EventTableEntry 8242: Group=, Trigger=conv1_buffer_upper_go_down 8243, Actions=[conv1_pallet_lifter_upper_up 8244], Comment=, ActivationMode=2, Cyclic=false
EventTableTriggerIO 8243: IOValue=[1], IRC5Controller=? -1, Operator=0, SignalSource=ALab_CellC_v1.0_4 5362
EventTableActionIO 8244: IOValue=[0], IRC5Controller=? -1, SignalTarget=ALab_CellC_v1.0_4 5362
EventTableEntry 8245: Group=, Trigger=conv1_buffer_upper_go_down 8246, Actions=[conv1_pallet_lifter_upper_up 8247], Comment=, ActivationMode=2, Cyclic=false
EventTableTriggerIO 8246: IOValue=[0], IRC5Controller=? -1, Operator=0, SignalSource=ALab_CellC_v1.0_4 5362
EventTableActionIO 8247: IOValue=[1], IRC5Controller=? -1, SignalTarget=ALab_CellC_v1.0_4 5362
EventTableEntry 8248: Group=, Trigger=conv1_buffer_upper_go_down 8249, Actions=[conv1_pallet_lifter_upper_down 8250], Comment=, ActivationMode=2, Cyclic=false
EventTableTriggerIO 8249: IOValue=[0], IRC5Controller=? -1, Operator=0, SignalSource=ALab_CellC_v1.0_4 5362
EventTableActionIO 8250: IOValue=[0], IRC5Controller=? -1, SignalTarget=ALab_CellC_v1.0_4 5362
EventTableEntry 8251: Group=, Trigger=conv1_buffer_upper_go_down 8252, Actions=[conv1_pallet_lifter_upper_down 8253], Comment=, ActivationMode=2, Cyclic=false
EventTableTriggerIO 8252: IOValue=[1], IRC5Controller=? -1, Operator=0, SignalSource=ALab_CellC_v1.0_4 5362
EventTableActionIO 8253: IOValue=[1], IRC5Controller=? -1, SignalTarget=ALab_CellC_v1.0_4 5362
EventTableEntry 8254: Group=, Trigger=conv1_buffer_lower_go_up 8255, Actions=[conv1_pallet_lifter_lower_down 8256], Comment=, ActivationMode=2, Cyclic=false
EventTableTriggerIO 8255: IOValue=[0], IRC5Controller=? -1, Operator=0, SignalSource=ALab_CellC_v1.0_4 5362
EventTableActionIO 8256: IOValue=[1], IRC5Controller=? -1, SignalTarget=ALab_CellC_v1.0_4 5362
EventTableEntry 8257: Group=, Trigger=conv1_buffer_lower_go_up 8258, Actions=[conv1_pallet_lifter_lower_down 8259], Comment=, ActivationMode=2, Cyclic=false
EventTableTriggerIO 8258: IOValue=[1], IRC5Controller=? -1, Operator=0, SignalSource=ALab_CellC_v1.0_4 5362
EventTableActionIO 8259: IOValue=[0], IRC5Controller=? -1, SignalTarget=ALab_CellC_v1.0_4 5362
EventTableEntry 8260: Group=, Trigger=conv2_buffer_horizontal_move 8261, Actions=[conv2_pallet_lifter_in 8262], Comment=, ActivationMode=2, Cyclic=false
EventTableTriggerIO 8261: IOValue=[1], IRC5Controller=? -1, Operator=0, SignalSource=ALab_CellC_v1.0_4 5362
EventTableActionIO 8262: IOValue=[1], IRC5Controller=? -1, SignalTarget=ALab_CellC_v1.0_4 5362
EventTableEntry 8263: Group=, Trigger=conv2_buffer_horizontal_move 8264, Actions=[conv2_pallet_lifter_in 8265], Comment=, ActivationMode=2, Cyclic=false
EventTableTriggerIO 8264: IOValue=[0], IRC5Controller=? -1, Operator=0, SignalSource=ALab_CellC_v1.0_4 5362
EventTableActionIO 8265: IOValue=[0], IRC5Controller=? -1, SignalTarget=ALab_CellC_v1.0_4 5362
EventTableEntry 8266: Group=, Trigger=conv2_buffer_horizontal_move 8267, Actions=[conv2_pallet_lifter_out 8268], Comment=, ActivationMode=2, Cyclic=false
EventTableTriggerIO 8267: IOValue=[0], IRC5Controller=? -1, Operator=0, SignalSource=ALab_CellC_v1.0_4 5362
EventTableActionIO 8268: IOValue=[1], IRC5Controller=? -1, SignalTarget=ALab_CellC_v1.0_4 5362
EventTableEntry 8269: Group=, Trigger=conv2_buffer_horizontal_move 8270, Actions=[conv2_pallet_lifter_out 8271], Comment=, ActivationMode=2, Cyclic=false
EventTableTriggerIO 8270: IOValue=[1], IRC5Controller=? -1, Operator=0, SignalSource=ALab_CellC_v1.0_4 5362
EventTableActionIO 8271: IOValue=[0], IRC5Controller=? -1, SignalTarget=ALab_CellC_v1.0_4 5362
EventTableEntry 8272: Group=, Trigger=conv2_buffer_lower_vertical_move 8273, Actions=[conv2_pallet_lifter_lower_down 8274], Comment=, ActivationMode=2, Cyclic=false
EventTableTriggerIO 8273: IOValue=[1], IRC5Controller=? -1, Operator=0, SignalSource=ALab_CellC_v1.0_4 5362
EventTableActionIO 8274: IOValue=[0], IRC5Controller=? -1, SignalTarget=ALab_CellC_v1.0_4 5362
EventTableEntry 8275: Group=, Trigger=conv2_buffer_lower_vertical_move 8276, Actions=[conv2_pallet_lifter_lower_down 8277], Comment=, ActivationMode=2, Cyclic=false
EventTableTriggerIO 8276: IOValue=[0], IRC5Controller=? -1, Operator=0, SignalSource=ALab_CellC_v1.0_4 5362
EventTableActionIO 8277: IOValue=[1], IRC5Controller=? -1, SignalTarget=ALab_CellC_v1.0_4 5362
EventTableEntry 8278: Group=, Trigger=conv2_buffer_upper_vertical_move 8279, Actions=[conv2_pallet_lifter_upper_up 8280], Comment=, ActivationMode=2, Cyclic=false
EventTableTriggerIO 8279: IOValue=[0], IRC5Controller=? -1, Operator=0, SignalSource=ALab_CellC_v1.0_4 5362
EventTableActionIO 8280: IOValue=[1], IRC5Controller=? -1, SignalTarget=ALab_CellC_v1.0_4 5362
EventTableEntry 8281: Group=, Trigger=conv2_buffer_upper_vertical_move 8282, Actions=[conv2_pallet_lifter_upper_up 8283], Comment=, ActivationMode=2, Cyclic=false
EventTableTriggerIO 8282: IOValue=[1], IRC5Controller=? -1, Operator=0, SignalSource=ALab_CellC_v1.0_4 5362
EventTableActionIO 8283: IOValue=[0], IRC5Controller=? -1, SignalTarget=ALab_CellC_v1.0_4 5362
EventTableEntry 8284: Group=, Trigger=conv2_buffer_upper_vertical_move 8285, Actions=[conv2_pallet_lifter_upper_down 8286], Comment=, ActivationMode=2, Cyclic=false
EventTableTriggerIO 8285: IOValue=[1], IRC5Controller=? -1, Operator=0, SignalSource=ALab_CellC_v1.0_4 5362
EventTableActionIO 8286: IOValue=[1], IRC5Controller=? -1, SignalTarget=ALab_CellC_v1.0_4 5362
EventTableEntry 8287: Group=, Trigger=conv2_buffer_upper_vertical_move 8288, Actions=[conv2_pallet_lifter_upper_down 8289], Comment=, ActivationMode=2, Cyclic=false
EventTableTriggerIO 8288: IOValue=[0], IRC5Controller=? -1, Operator=0, SignalSource=ALab_CellC_v1.0_4 5362
EventTableActionIO 8289: IOValue=[0], IRC5Controller=? -1, SignalTarget=ALab_CellC_v1.0_4 5362
EventTableTriggerIO 8290: IOValue=[-1], IRC5Controller=? -1, Operator=0, SignalSource=LCFA_profile 1
EventTableTriggerLogic 8291: layoutX=22, layoutY=19, Operand1=conv2_buffer_horizontal_move 8292, Operand2=? -1, Operator=2, Delay=1000
EventTableTriggerIO 8292: IOValue=[-1], IRC5Controller=? -1, Operator=0, SignalSource=ALab_CellC_v1.0_4 5362
EventTableEntry 8293: Group=, Trigger=pallet1.1 8294, Actions=[pickpallet4 8295], Comment=, ActivationMode=2, Cyclic=false
EventTableTriggerIO 8294: IOValue=[1], IRC5Controller=? -1, Operator=0, SignalSource=LCFA_profile 1
EventTableActionIO 8295: IOValue=[0], IRC5Controller=? -1, SignalTarget=LCFA_profile 1
EventTableEntry 8296: Group=, Trigger=pallet1.1 8297, Actions=[Pallet2.6 8298], Comment=, ActivationMode=2, Cyclic=false
EventTableTriggerIO 8297: IOValue=[1], IRC5Controller=? -1, Operator=0, SignalSource=LCFA_profile 1
EventTableActionIO 8298: IOValue=[0], IRC5Controller=? -1, SignalTarget=LCFA_profile 1
EventTableTriggerLogic 8357: layoutX=167, layoutY=76, Operand1=AND 4076, Operand2=AND 4081, Operator=0, Delay=1000
EventTableTriggerLogic 8358: layoutX=194, layoutY=70, Operand1=AND 4088, Operand2=AND 4093, Operator=0, Delay=1000
EventTableTriggerLogic 8359: layoutX=181, layoutY=88, Operand1=AND 4100, Operand2=AND 4105, Operator=0, Delay=1000
EventTableTriggerLogic 8360: layoutX=165, layoutY=70, Operand1=AND 4112, Operand2=AND 4117, Operator=0, Delay=1000
EventTableTriggerLogic 8361: layoutX=217, layoutY=77, Operand1=AND 4123, Operand2=AND 4127, Operator=0, Delay=1000
EventTableTriggerLogic 8362: layoutX=168, layoutY=84, Operand1=AND 4135, Operand2=AND 4139, Operator=0, Delay=1000
EventTableTriggerLogic 8363: layoutX=219, layoutY=73, Operand1=AND 4146, Operand2=AND 4150, Operator=0, Delay=1000
EventTableTriggerLogic 8364: layoutX=203, layoutY=67, Operand1=AND 4157, Operand2=AND 4161, Operator=0, Delay=1000
EventTableTriggerLogic 8365: layoutX=220, layoutY=69, Operand1=AND 4167, Operand2=AND 4171, Operator=0, Delay=1000
EventTableTriggerLogic 8366: layoutX=243, layoutY=55, Operand1=AND 4179, Operand2=AND 4183, Operator=0, Delay=1000
EventTableTriggerLogic 8367: layoutX=204, layoutY=112, Operand1=AND 4190, Operand2=AND 4194, Operator=0, Delay=1000
EventTableTriggerLogic 8368: layoutX=245, layoutY=97, Operand1=AND 4201, Operand2=AND 4205, Operator=0, Delay=1000
EventTableTriggerLogic 8369: layoutX=234, layoutY=61, Operand1=AND 4211, Operand2=AND 4214, Operator=0, Delay=1000
EventTableTriggerLogic 8370: layoutX=192, layoutY=87, Operand1=AND 4222, Operand2=AND 4225, Operator=0, Delay=1000
EventTableTriggerLogic 8371: layoutX=212, layoutY=64, Operand1=AND 4232, Operand2=AND 4235, Operator=0, Delay=1000
EventTableTriggerLogic 8372: layoutX=160, layoutY=73, Operand1=AND 4242, Operand2=AND 4245, Operator=0, Delay=1000
EventTableTriggerLogic 8373: layoutX=153, layoutY=73, Operand1=AND 4264, Operand2=NOT 4269, Operator=0, Delay=1000
EventTableTriggerLogic 8374: layoutX=133, layoutY=81, Operand1=AND 4274, Operand2=conv1_buffer_upper_go_down 6332, Operator=0, Delay=1000
EventTableTriggerLogic 8375: layoutX=184, layoutY=91, Operand1=AND 4283, Operand2=NOT 4287, Operator=0, Delay=1000
EventTableTriggerLogic 8376: layoutX=211, layoutY=90, Operand1=AND 4292, Operand2=conv1_buffer_upper_go_down 6282, Operator=0, Delay=1000
EventTableTriggerLogic 8377: layoutX=226, layoutY=110, Operand1=AND 4300, Operand2=NOT 4304, Operator=0, Delay=1000
EventTableTriggerLogic 8378: layoutX=164, layoutY=68, Operand1=AND 4309, Operand2=conv1_buffer_upper_go_down 6288, Operator=0, Delay=1000
EventTableTriggerLogic 8379: layoutX=161, layoutY=63, Operand1=AND 4317, Operand2=NOT 4320, Operator=0, Delay=1000
EventTableTriggerLogic 8380: layoutX=174, layoutY=87, Operand1=AND 4325, Operand2=conv1_buffer_upper_go_down 6294, Operator=0, Delay=1000
EventTableTriggerLogic 8381: layoutX=148, layoutY=98, Operand1=AND 4332, Operand2=NOT 4337, Operator=0, Delay=1000
EventTableTriggerLogic 8382: layoutX=206, layoutY=74, Operand1=AND 4342, Operand2=conv2_buffer_upper_vertical_move 6300, Operator=0, Delay=1000
EventTableTriggerLogic 8383: layoutX=195, layoutY=82, Operand1=AND 4351, Operand2=NOT 4355, Operator=0, Delay=1000
EventTableTriggerLogic 8384: layoutX=193, layoutY=94, Operand1=AND 4360, Operand2=conv2_buffer_upper_vertical_move 6306, Operator=0, Delay=1000
EventTableTriggerLogic 8385: layoutX=210, layoutY=27, Operand1=conv2_buffer_horizontal_move 6309, Operand2=AND 4369, Operator=0, Delay=1000
EventTableTriggerLogic 8386: layoutX=233, layoutY=95, Operand1=AND 4377, Operand2=conv2_buffer_upper_vertical_move 6312, Operator=0, Delay=1000
EventTableTriggerLogic 8387: layoutX=102, layoutY=69, Operand1=AND 4385, Operand2=NOT 4388, Operator=0, Delay=1000
EventTableTriggerLogic 8388: layoutX=97, layoutY=92, Operand1=AND 4393, Operand2=conv2_buffer_upper_vertical_move 6318, Operator=0, Delay=1000
EventTableTriggerLogic 8389: layoutX=96, layoutY=16, Operand1=cellC_pallet_holder 7125, Operand2=cellC_pallet_stopper 7126, Operator=0, Delay=1000
EventTableTriggerLogic 8390: layoutX=142, layoutY=32, Operand1=NOT 7128, Operand2=cellC_pallet_stopper 7127, Operator=0, Delay=1000
EventTableTriggerLogic 8391: layoutX=51, layoutY=46, Operand1=NOT 7130, Operand2=NOT 7132, Operator=0, Delay=1000
EventTableTriggerLogic 8392: layoutX=107, layoutY=60, Operand1=cellC_pallet_holder 7134, Operand2=NOT 7135, Operator=0, Delay=1000
EventTableTriggerIO 8394: IOValue=[1], IRC5Controller=? -1, Operator=0, SignalSource=ALab_CellC_v1.0_4 5362
EventTableTriggerLogic 8407: layoutX=184, layoutY=128, Operand1=AND 6402, Operand2=AND 6408, Operator=0, Delay=1000
EventTableTriggerLogic 8408: layoutX=231, layoutY=144, Operand1=AND 6416, Operand2=pallet1 6426, Operator=0, Delay=1000
EventTableTriggerLogic 8409: layoutX=251, layoutY=143, Operand1=AND 8115, Operand2=pallet3.1 8114, Operator=0, Delay=1000
EventTableTriggerLogic 8410: layoutX=62, layoutY=38, Operand1=pallet2 8126, Operand2=cellC_slider_horizontal_move 8125, Operator=0, Delay=1000
EventTableTriggerLogic 8411: layoutX=133, layoutY=37, Operand1=pallet3 6451, Operand2=pose6 6452, Operator=0, Delay=1000
EventTableTriggerLogic 8412: layoutX=61, layoutY=50, Operand1=pallet3.2 6456, Operand2=pose3 6457, Operator=0, Delay=1000
EventTableTriggerLogic 8413: layoutX=131, layoutY=52, Operand1=pickpallet1 6461, Operand2=pose7 6462, Operator=0, Delay=1000
EventTableTriggerLogic 8414: layoutX=8, layoutY=16, Operand1=pickpallet2 6466, Operand2=pose13 6467, Operator=0, Delay=1000
EventTableTriggerLogic 8415: layoutX=232, layoutY=117, Operand1=AND 6471, Operand2=pallet4 6481, Operator=0, Delay=1000
EventTableTriggerLogic 8416: layoutX=237, layoutY=122, Operand1=AND 6485, Operand2=conv2_buffer_stopper 6492, Operator=0, Delay=1000
EventTableTriggerLogic 8417: layoutX=240, layoutY=90, Operand1=AND 6496, Operand2=AND 6500, Operator=0, Delay=1000
EventTableTriggerLogic 8418: layoutX=80, layoutY=49, Operand1=pallet5.1 6513, Operand2=conv2_outer_lifter 6514, Operator=0, Delay=1000
EventTableTriggerIO 8419: IOValue=[1], IRC5Controller=? -1, Operator=0, SignalSource=LCFA_profile 1
EventTableTriggerIO 8420: IOValue=[1], IRC5Controller=? -1, Operator=0, SignalSource=LCFA_profile 1
EventTableTriggerIO 8421: IOValue=[1], IRC5Controller=? -1, Operator=0, SignalSource=LCFA_profile 1
EventTableTriggerIO 8422: IOValue=[1], IRC5Controller=? -1, Operator=0, SignalSource=LCFA_profile 1
EventTableTriggerIO 8423: IOValue=[1], IRC5Controller=? -1, Operator=0, SignalSource=LCFA_profile 1
EventTableTriggerIO 8424: IOValue=[1], IRC5Controller=? -1, Operator=0, SignalSource=LCFA_profile 1
EventTableTriggerIO 8425: IOValue=[1], IRC5Controller=? -1, Operator=0, SignalSource=LCFA_profile 1
EventTableTriggerIO 8426: IOValue=[1], IRC5Controller=? -1, Operator=0, SignalSource=LCFA_profile 1
EventTableTriggerIO 8427: IOValue=[1], IRC5Controller=? -1, Operator=0, SignalSource=LCFA_profile 1
EventTableTriggerIO 8428: IOValue=[1], IRC5Controller=? -1, Operator=0, SignalSource=LCFA_profile 1
EventTableTriggerIO 8429: IOValue=[0], IRC5Controller=? -1, Operator=0, SignalSource=ALab_CellC_v1.0_4 5362
EventTableTriggerIO 8430: IOValue=[1], IRC5Controller=? -1, Operator=0, SignalSource=ALab_CellC_v1.0_4 5362
EventTableTriggerIO 8431: IOValue=[0], IRC5Controller=? -1, Operator=0, SignalSource=ALab_CellC_v1.0_4 5362
EventTableTriggerIO 8432: IOValue=[1], IRC5Controller=? -1, Operator=0, SignalSource=ALab_CellC_v1.0_4 5362
EventTableTriggerIO 8433: IOValue=[1], IRC5Controller=? -1, Operator=0, SignalSource=ALab_CellC_v1.0_4 5362
EventTableTriggerIO 8434: IOValue=[0], IRC5Controller=? -1, Operator=0, SignalSource=ALab_CellC_v1.0_4 5362
EventTableTriggerIO 8435: IOValue=[0], IRC5Controller=? -1, Operator=0, SignalSource=ALab_CellC_v1.0_4 5362
EventTableTriggerIO 8436: IOValue=[1], IRC5Controller=? -1, Operator=0, SignalSource=ALab_CellC_v1.0_4 5362
EventTableTriggerIO 8437: IOValue=[1], IRC5Controller=? -1, Operator=0, SignalSource=ALab_CellC_v1.0_4 5362
EventTableTriggerIO 8438: IOValue=[0], IRC5Controller=? -1, Operator=0, SignalSource=ALab_CellC_v1.0_4 5362
EventTableTriggerIO 8439: IOValue=[1], IRC5Controller=? -1, Operator=0, SignalSource=ALab_CellC_v1.0_4 5362
EventTableTriggerIO 8440: IOValue=[0], IRC5Controller=? -1, Operator=0, SignalSource=ALab_CellC_v1.0_4 5362
EventTableTriggerIO 8441: IOValue=[0], IRC5Controller=? -1, Operator=0, SignalSource=ALab_CellC_v1.0_4 5362
EventTableTriggerIO 8442: IOValue=[1], IRC5Controller=? -1, Operator=0, SignalSource=ALab_CellC_v1.0_4 5362
EventTableTriggerIO 8443: IOValue=[1], IRC5Controller=? -1, Operator=0, SignalSource=ALab_CellC_v1.0_4 5362
EventTableTriggerIO 8444: IOValue=[0], IRC5Controller=? -1, Operator=0, SignalSource=ALab_CellC_v1.0_4 5362
EventTableTriggerIO 8445: IOValue=[0], IRC5Controller=? -1, Operator=0, SignalSource=ALab_CellC_v1.0_4 5362
EventTableTriggerIO 8446: IOValue=[1], IRC5Controller=? -1, Operator=0, SignalSource=ALab_CellC_v1.0_4 5362
EventTableTriggerIO 8447: IOValue=[1], IRC5Controller=? -1, Operator=0, SignalSource=ALab_CellC_v1.0_4 5362
EventTableTriggerIO 8448: IOValue=[0], IRC5Controller=? -1, Operator=0, SignalSource=ALab_CellC_v1.0_4 5362
EventTableTriggerIO 8449: IOValue=[1], IRC5Controller=? -1, Operator=0, SignalSource=LCFA_profile 1
EventTableTriggerIO 8450: IOValue=[1], IRC5Controller=? -1, Operator=0, SignalSource=LCFA_profile 1
EventTableTriggerIO 8451: IOValue=[1], IRC5Controller=? -1, Operator=0, SignalSource=LCFA_profile 1
EventTableTriggerIO 8452: IOValue=[1], IRC5Controller=? -1, Operator=0, SignalSource=LCFA_profile 1
EventTableTriggerIO 8453: IOValue=[1], IRC5Controller=? -1, Operator=0, SignalSource=ALab_CellC_v1.0_4 5362
EventTableTriggerIO 8454: IOValue=[0], IRC5Controller=? -1, Operator=0, SignalSource=ALab_CellC_v1.0_4 5362
EventTableTriggerIO 8455: IOValue=[1], IRC5Controller=? -1, Operator=0, SignalSource=LCFA_profile 1
EventTableTriggerIO 8456: IOValue=[1], IRC5Controller=? -1, Operator=0, SignalSource=LCFA_profile 1
EventTableTriggerIO 8457: IOValue=[1], IRC5Controller=? -1, Operator=0, SignalSource=LCFA_profile 1
EventTableTriggerIO 8458: IOValue=[1], IRC5Controller=? -1, Operator=0, SignalSource=LCFA_profile 1
EventTableTriggerIO 8459: IOValue=[1], IRC5Controller=? -1, Operator=0, SignalSource=ALab_CellC_v1.0_4 5362
EventTableTriggerIO 8460: IOValue=[0], IRC5Controller=? -1, Operator=0, SignalSource=ALab_CellC_v1.0_4 5362
EventTableTriggerIO 8461: IOValue=[1], IRC5Controller=? -1, Operator=0, SignalSource=ALab_CellC_v1.0_4 5362
EventTableTriggerIO 8462: IOValue=[0], IRC5Controller=? -1, Operator=0, SignalSource=ALab_CellC_v1.0_4 5362
EventTableTriggerIO 8463: IOValue=[0], IRC5Controller=? -1, Operator=0, SignalSource=ALab_CellC_v1.0_4 5362
EventTableTriggerIO 8464: IOValue=[1], IRC5Controller=? -1, Operator=0, SignalSource=ALab_CellC_v1.0_4 5362
EventTableTriggerIO 8465: IOValue=[1], IRC5Controller=? -1, Operator=0, SignalSource=ALab_CellC_v1.0_4 5362
EventTableTriggerIO 8466: IOValue=[0], IRC5Controller=? -1, Operator=0, SignalSource=ALab_CellC_v1.0_4 5362
EventTableTriggerIO 8471: IOValue=[1], IRC5Controller=? -1, Operator=0, SignalSource=LCFA_profile 1
EventTableTriggerIO 8472: IOValue=[1], IRC5Controller=? -1, Operator=0, SignalSource=LCFA_profile 1
EventTableTriggerIO 8473: IOValue=[1], IRC5Controller=? -1, Operator=0, SignalSource=LCFA_profile 1
EventTableTriggerLogic 8474: layoutX=150, layoutY=90, Operand1=AND 6770, Operand2=conv2_motor_s1 6766, Operator=0, Delay=1000
EventTableTriggerIO 8475: IOValue=[1], IRC5Controller=? -1, Operator=0, SignalSource=LCFA_profile 1
EventTableTriggerIO 8476: IOValue=[1], IRC5Controller=? -1, Operator=0, SignalSource=LCFA_profile 1
EventTableTriggerIO 8477: IOValue=[1], IRC5Controller=? -1, Operator=0, SignalSource=LCFA_profile 1
EventTableTriggerIO 8478: IOValue=[1], IRC5Controller=? -1, Operator=0, SignalSource=LCFA_profile 1
EventTableTriggerIO 8479: IOValue=[1], IRC5Controller=? -1, Operator=0, SignalSource=LCFA_profile 1
EventTableTriggerIO 8480: IOValue=[1], IRC5Controller=? -1, Operator=0, SignalSource=LCFA_profile 1
EventTableTriggerIO 8481: IOValue=[1], IRC5Controller=? -1, Operator=0, SignalSource=LCFA_profile 1
EventTableTriggerIO 8482: IOValue=[1], IRC5Controller=? -1, Operator=0, SignalSource=LCFA_profile 1
EventTableTriggerIO 8483: IOValue=[1], IRC5Controller=? -1, Operator=0, SignalSource=LCFA_profile 1
EventTableTriggerIO 8484: IOValue=[1], IRC5Controller=? -1, Operator=0, SignalSource=LCFA_profile 1
EventTableTriggerIO 8485: IOValue=[1], IRC5Controller=? -1, Operator=0, SignalSource=LCFA_profile 1
EventTableTriggerIO 8486: IOValue=[1], IRC5Controller=? -1, Operator=0, SignalSource=LCFA_profile 1
EventTableTriggerLogic 8487: layoutX=155, layoutY=137, Operand1=AND 6751, Operand2=NOT 6755, Operator=0, Delay=1000
EventTableTriggerIO 8488: IOValue=[1], IRC5Controller=? -1, Operator=0, SignalSource=LCFA_profile 1
EventTableTriggerIO 8489: IOValue=[1], IRC5Controller=? -1, Operator=0, SignalSource=LCFA_profile 1
EventTableTriggerLogic 8490: layoutX=48, layoutY=41, Operand1=pallet1.1 6778, Operand2=PalletIO00 6779, Operator=0, Delay=1000
EventTableTriggerIO 8491: IOValue=[1], IRC5Controller=? -1, Operator=0, SignalSource=LCFA_profile 1
EventTableTriggerIO 8492: IOValue=[1], IRC5Controller=? -1, Operator=0, SignalSource=ALab_CellC_v1.0_4 5362
EventTableTriggerIO 8493: IOValue=[0], IRC5Controller=? -1, Operator=0, SignalSource=ALab_CellC_v1.0_4 5362
EventTableTriggerLogic 8494: layoutX=103, layoutY=47, Operand1=NOT 8291, Operand2=pallet5 8290, Operator=0, Delay=1000
EventTableTriggerLogic 8495: layoutX=79, layoutY=37, Operand1=Pallet5.3 8029, Operand2=conv2_buffer_upper_vertical_move 8133, Operator=0, Delay=1000
EventTableTriggerLogic 8496: layoutX=40, layoutY=37, Operand1=Pallet5.4 8035, Operand2=conv2_buffer_lower_vertical_move 8036, Operator=0, Delay=1000
EventTableTriggerLogic 8497: layoutX=103, layoutY=47, Operand1=conv2_buffer_horizontal_move 8134, Operand2=Pallet5.7 8040, Operator=0, Delay=1000
EventTableTriggerLogic 8498: layoutX=54, layoutY=45, Operand1=NOT 8135, Operand2=Pallet5.6 8046, Operator=0, Delay=1000
EventTableTriggerLogic 8499: layoutX=108, layoutY=46, Operand1=NOT 8052, Operand2=Pallet5.5 8051, Operator=0, Delay=1000
EventTableTriggerIO 8500: IOValue=[1], IRC5Controller=? -1, Operator=0, SignalSource=LCFA_profile 1
EventTableTriggerIO 8501: IOValue=[1], IRC5Controller=? -1, Operator=0, SignalSource=LCFA_profile 1
EventTableTriggerIO 8502: IOValue=[1], IRC5Controller=? -1, Operator=0, SignalSource=LCFA_profile 1
EventTableTriggerIO 8503: IOValue=[1], IRC5Controller=? -1, Operator=0, SignalSource=LCFA_profile 1
EventTableTriggerIO 8504: IOValue=[1], IRC5Controller=? -1, Operator=0, SignalSource=LCFA_profile 1
EventTableTriggerIO 8505: IOValue=[1], IRC5Controller=? -1, Operator=0, SignalSource=LCFA_profile 1
EventTableTriggerIO 8506: IOValue=[1], IRC5Controller=? -1, Operator=0, SignalSource=LCFA_profile 1
EventTableTriggerIO 8507: IOValue=[1], IRC5Controller=? -1, Operator=0, SignalSource=LCFA_profile 1
EventTableTriggerIO 8508: IOValue=[1], IRC5Controller=? -1, Operator=0, SignalSource=LCFA_profile 1
EventTableTriggerIO 8509: IOValue=[1], IRC5Controller=? -1, Operator=0, SignalSource=LCFA_profile 1
EventTableTriggerIO 8510: IOValue=[1], IRC5Controller=? -1, Operator=0, SignalSource=LCFA_profile 1
EventTableTriggerIO 8511: IOValue=[1], IRC5Controller=? -1, Operator=0, SignalSource=LCFA_profile 1
EventTableTriggerIO 8512: IOValue=[1], IRC5Controller=? -1, Operator=0, SignalSource=LCFA_profile 1
EventTableTriggerIO 8513: IOValue=[1], IRC5Controller=? -1, Operator=0, SignalSource=LCFA_profile 1
EventTableTriggerIO 8514: IOValue=[1], IRC5Controller=? -1, Operator=0, SignalSource=LCFA_profile 1
EventTableTriggerIO 8515: IOValue=[1], IRC5Controller=? -1, Operator=0, SignalSource=LCFA_profile 1
EventTableTriggerIO 8516: IOValue=[1], IRC5Controller=? -1, Operator=0, SignalSource=LCFA_profile 1
EventTableTriggerLogic 8517: layoutX=99, layoutY=32, Operand1=Pallet2.1 8141, Operand2=NOT 8139, Operator=0, Delay=1000
EventTableTriggerLogic 8518: layoutX=181, layoutY=52, Operand1=conv1_buffer_upper_go_down 8146, Operand2=Pallet2.2 8145, Operator=0, Delay=1000
EventTableTriggerLogic 8519: layoutX=48, layoutY=51, Operand1=Pallet2.3 8150, Operand2=conv1_buffer_lower_go_up 8151, Operator=0, Delay=1000
EventTableTriggerLogic 8520: layoutX=67, layoutY=33, Operand1=pallet2 8155, Operand2=NOT 8156, Operator=0, Delay=1000
EventTableTriggerLogic 8521: layoutX=102, layoutY=29, Operand1=Pallet2.4 8161, Operand2=NOT 8162, Operator=0, Delay=1000
EventTableTriggerLogic 8522: layoutX=102, layoutY=23, Operand1=Pallet2.5 8167, Operand2=NOT 8168, Operator=0, Delay=1000
EventTableTriggerIO 8523: IOValue=[1], IRC5Controller=? -1, Operator=0, SignalSource=LCFA_profile 1
EventTableTriggerIO 8524: IOValue=[1], IRC5Controller=? -1, Operator=0, SignalSource=LCFA_profile 1
EventTableTriggerIO 8525: IOValue=[1], IRC5Controller=? -1, Operator=0, SignalSource=LCFA_profile 1
EventTableTriggerIO 8526: IOValue=[1], IRC5Controller=? -1, Operator=0, SignalSource=LCFA_profile 1
EventTableTriggerIO 8527: IOValue=[1], IRC5Controller=? -1, Operator=0, SignalSource=LCFA_profile 1
EventTableTriggerIO 8528: IOValue=[1], IRC5Controller=? -1, Operator=0, SignalSource=LCFA_profile 1
EventTableTriggerIO 8529: IOValue=[1], IRC5Controller=? -1, Operator=0, SignalSource=LCFA_profile 1
EventTableTriggerIO 8530: IOValue=[1], IRC5Controller=? -1, Operator=0, SignalSource=LCFA_profile 1
EventTableTriggerIO 8531: IOValue=[1], IRC5Controller=? -1, Operator=0, SignalSource=LCFA_profile 1
EventTableTriggerIO 8532: IOValue=[1], IRC5Controller=? -1, Operator=0, SignalSource=LCFA_profile 1
EventTableTriggerIO 8533: IOValue=[1], IRC5Controller=? -1, Operator=0, SignalSource=LCFA_profile 1
EventTableTriggerIO 8534: IOValue=[1], IRC5Controller=? -1, Operator=0, SignalSource=LCFA_profile 1
EventTableTriggerIO 8535: IOValue=[1], IRC5Controller=? -1, Operator=0, SignalSource=LCFA_profile 1
EventTableTriggerLogic 8536: layoutX=49, layoutY=26, Operand1=Pallet2.6 8213, Operand2=conv1_buffer_horizontal_open 8214, Operator=0, Delay=1000
EventTableTriggerIO 8537: IOValue=[1], IRC5Controller=? -1, Operator=0, SignalSource=LCFA_profile 1
EventTableTriggerIO 8538: IOValue=[1], IRC5Controller=? -1, Operator=0, SignalSource=LCFA_profile 1
EventTableTriggerIO 8539: IOValue=[1], IRC5Controller=? -1, Operator=0, SignalSource=LCFA_profile 1
EventTableTriggerIO 8540: IOValue=[1], IRC5Controller=? -1, Operator=0, SignalSource=LCFA_profile 1
EventTableTriggerIO 8541: IOValue=[1], IRC5Controller=? -1, Operator=0, SignalSource=LCFA_profile 1
EventTableTriggerIO 8542: IOValue=[1], IRC5Controller=? -1, Operator=0, SignalSource=ALab_CellC_v1.0_4 5362
EventTableTriggerIO 8543: IOValue=[0], IRC5Controller=? -1, Operator=0, SignalSource=ALab_CellC_v1.0_4 5362
EventTableTriggerIO 8544: IOValue=[1], IRC5Controller=? -1, Operator=0, SignalSource=ALab_CellC_v1.0_4 5362
EventTableTriggerIO 8545: IOValue=[0], IRC5Controller=? -1, Operator=0, SignalSource=ALab_CellC_v1.0_4 5362
EventTableTriggerIO 8546: IOValue=[1], IRC5Controller=? -1, Operator=0, SignalSource=ALab_CellC_v1.0_4 5362
EventTableTriggerIO 8547: IOValue=[0], IRC5Controller=? -1, Operator=0, SignalSource=ALab_CellC_v1.0_4 5362
EventTableTriggerIO 8548: IOValue=[0], IRC5Controller=? -1, Operator=0, SignalSource=ALab_CellC_v1.0_4 5362
EventTableTriggerIO 8549: IOValue=[1], IRC5Controller=? -1, Operator=0, SignalSource=ALab_CellC_v1.0_4 5362
EventTableTriggerIO 8550: IOValue=[0], IRC5Controller=? -1, Operator=0, SignalSource=ALab_CellC_v1.0_4 5362
EventTableTriggerIO 8551: IOValue=[1], IRC5Controller=? -1, Operator=0, SignalSource=ALab_CellC_v1.0_4 5362
EventTableTriggerIO 8552: IOValue=[1], IRC5Controller=? -1, Operator=0, SignalSource=ALab_CellC_v1.0_4 5362
EventTableTriggerIO 8553: IOValue=[0], IRC5Controller=? -1, Operator=0, SignalSource=ALab_CellC_v1.0_4 5362
EventTableTriggerIO 8554: IOValue=[0], IRC5Controller=? -1, Operator=0, SignalSource=ALab_CellC_v1.0_4 5362
EventTableTriggerIO 8555: IOValue=[1], IRC5Controller=? -1, Operator=0, SignalSource=ALab_CellC_v1.0_4 5362
EventTableTriggerIO 8556: IOValue=[1], IRC5Controller=? -1, Operator=0, SignalSource=ALab_CellC_v1.0_4 5362
EventTableTriggerIO 8557: IOValue=[0], IRC5Controller=? -1, Operator=0, SignalSource=ALab_CellC_v1.0_4 5362
EventTableTriggerIO 8558: IOValue=[0], IRC5Controller=? -1, Operator=0, SignalSource=ALab_CellC_v1.0_4 5362
EventTableTriggerIO 8559: IOValue=[1], IRC5Controller=? -1, Operator=0, SignalSource=ALab_CellC_v1.0_4 5362
EventTableTriggerIO 8560: IOValue=[1], IRC5Controller=? -1, Operator=0, SignalSource=ALab_CellC_v1.0_4 5362
EventTableTriggerIO 8561: IOValue=[0], IRC5Controller=? -1, Operator=0, SignalSource=ALab_CellC_v1.0_4 5362
EventTableTriggerIO 8562: IOValue=[1], IRC5Controller=? -1, Operator=0, SignalSource=LCFA_profile 1
EventTableTriggerIO 8563: IOValue=[1], IRC5Controller=? -1, Operator=0, SignalSource=LCFA_profile 1
EventTableEntry 8586: Group=, Trigger=Rob1_Gripper_set 8587, Actions=[EventTableActionMechanicalPose 8588], Comment=, ActivationMode=2, Cyclic=false
EventTableTriggerIO 8587: IOValue=[1], IRC5Controller=? -1, Operator=0, SignalSource=ALab_CellC_v1.0_4 5362
EventTableActionMechanicalPose 8588: VirtualSignal=, Mechanism=Gripper 8576, ToPoseName=ClosePose, VirtualSignalValue=[1]
EventTableEntry 8589: Group=, Trigger=Rob1_Gripper_set 8590, Actions=[EventTableActionMechanicalPose 8591], Comment=, ActivationMode=2, Cyclic=false
EventTableTriggerIO 8590: IOValue=[0], IRC5Controller=? -1, Operator=0, SignalSource=ALab_CellC_v1.0_4 5362
EventTableActionMechanicalPose 8591: VirtualSignal=, Mechanism=Gripper 8576, ToPoseName=ClosePose, VirtualSignalValue=[1]
EventTableEntry 8592: Group=, Trigger=Rob1_Gripper_reset 8593, Actions=[EventTableActionMechanicalPose 8594], Comment=, ActivationMode=2, Cyclic=false
EventTableTriggerIO 8593: IOValue=[1], IRC5Controller=? -1, Operator=0, SignalSource=ALab_CellC_v1.0_4 5362
EventTableActionMechanicalPose 8594: VirtualSignal=, Mechanism=Gripper 8576, ToPoseName=HomePosition, VirtualSignalValue=[1]
EventTableEntry 8595: Group=, Trigger=Rob1_Gripper_reset 8596, Actions=[EventTableActionMechanicalPose 8597], Comment=, ActivationMode=2, Cyclic=false
EventTableTriggerIO 8596: IOValue=[0], IRC5Controller=? -1, Operator=0, SignalSource=ALab_CellC_v1.0_4 5362
EventTableActionMechanicalPose 8597: VirtualSignal=, Mechanism=Gripper 8576, ToPoseName=HomePosition, VirtualSignalValue=[1]
EventTableTriggerLogic 8820: layoutX=167, layoutY=76, Operand1=AND 4076, Operand2=AND 4081, Operator=0, Delay=1000
EventTableTriggerLogic 8821: layoutX=194, layoutY=70, Operand1=AND 4088, Operand2=AND 4093, Operator=0, Delay=1000
EventTableTriggerLogic 8822: layoutX=181, layoutY=88, Operand1=AND 4100, Operand2=AND 4105, Operator=0, Delay=1000
EventTableTriggerLogic 8823: layoutX=165, layoutY=70, Operand1=AND 4112, Operand2=AND 4117, Operator=0, Delay=1000
EventTableTriggerLogic 8824: layoutX=217, layoutY=77, Operand1=AND 4123, Operand2=AND 4127, Operator=0, Delay=1000
EventTableTriggerLogic 8825: layoutX=168, layoutY=84, Operand1=AND 4135, Operand2=AND 4139, Operator=0, Delay=1000
EventTableTriggerLogic 8826: layoutX=219, layoutY=73, Operand1=AND 4146, Operand2=AND 4150, Operator=0, Delay=1000
EventTableTriggerLogic 8827: layoutX=203, layoutY=67, Operand1=AND 4157, Operand2=AND 4161, Operator=0, Delay=1000
EventTableTriggerLogic 8828: layoutX=220, layoutY=69, Operand1=AND 4167, Operand2=AND 4171, Operator=0, Delay=1000
EventTableTriggerLogic 8829: layoutX=243, layoutY=55, Operand1=AND 4179, Operand2=AND 4183, Operator=0, Delay=1000
EventTableTriggerLogic 8830: layoutX=204, layoutY=112, Operand1=AND 4190, Operand2=AND 4194, Operator=0, Delay=1000
EventTableTriggerLogic 8831: layoutX=245, layoutY=97, Operand1=AND 4201, Operand2=AND 4205, Operator=0, Delay=1000
EventTableTriggerLogic 8832: layoutX=234, layoutY=61, Operand1=AND 4211, Operand2=AND 4214, Operator=0, Delay=1000
EventTableTriggerLogic 8833: layoutX=192, layoutY=87, Operand1=AND 4222, Operand2=AND 4225, Operator=0, Delay=1000
EventTableTriggerLogic 8834: layoutX=212, layoutY=64, Operand1=AND 4232, Operand2=AND 4235, Operator=0, Delay=1000
EventTableTriggerLogic 8835: layoutX=160, layoutY=73, Operand1=AND 4242, Operand2=AND 4245, Operator=0, Delay=1000
EventTableTriggerLogic 8836: layoutX=153, layoutY=73, Operand1=AND 4264, Operand2=NOT 4269, Operator=0, Delay=1000
EventTableTriggerLogic 8837: layoutX=133, layoutY=81, Operand1=AND 4274, Operand2=conv1_buffer_upper_go_down 6332, Operator=0, Delay=1000
EventTableTriggerLogic 8838: layoutX=184, layoutY=91, Operand1=AND 4283, Operand2=NOT 4287, Operator=0, Delay=1000
EventTableTriggerLogic 8839: layoutX=211, layoutY=90, Operand1=AND 4292, Operand2=conv1_buffer_upper_go_down 6282, Operator=0, Delay=1000
EventTableTriggerLogic 8840: layoutX=226, layoutY=110, Operand1=AND 4300, Operand2=NOT 4304, Operator=0, Delay=1000
EventTableTriggerLogic 8841: layoutX=164, layoutY=68, Operand1=AND 4309, Operand2=conv1_buffer_upper_go_down 6288, Operator=0, Delay=1000
EventTableTriggerLogic 8842: layoutX=161, layoutY=63, Operand1=AND 4317, Operand2=NOT 4320, Operator=0, Delay=1000
EventTableTriggerLogic 8843: layoutX=174, layoutY=87, Operand1=AND 4325, Operand2=conv1_buffer_upper_go_down 6294, Operator=0, Delay=1000
EventTableTriggerLogic 8844: layoutX=148, layoutY=98, Operand1=AND 4332, Operand2=NOT 4337, Operator=0, Delay=1000
EventTableTriggerLogic 8845: layoutX=206, layoutY=74, Operand1=AND 4342, Operand2=conv2_buffer_upper_vertical_move 6300, Operator=0, Delay=1000
EventTableTriggerLogic 8846: layoutX=195, layoutY=82, Operand1=AND 4351, Operand2=NOT 4355, Operator=0, Delay=1000
EventTableTriggerLogic 8847: layoutX=193, layoutY=94, Operand1=AND 4360, Operand2=conv2_buffer_upper_vertical_move 6306, Operator=0, Delay=1000
EventTableTriggerLogic 8848: layoutX=210, layoutY=27, Operand1=conv2_buffer_horizontal_move 6309, Operand2=AND 4369, Operator=0, Delay=1000
EventTableTriggerLogic 8849: layoutX=233, layoutY=95, Operand1=AND 4377, Operand2=conv2_buffer_upper_vertical_move 6312, Operator=0, Delay=1000
EventTableTriggerLogic 8850: layoutX=102, layoutY=69, Operand1=AND 4385, Operand2=NOT 4388, Operator=0, Delay=1000
EventTableTriggerLogic 8851: layoutX=97, layoutY=92, Operand1=AND 4393, Operand2=conv2_buffer_upper_vertical_move 6318, Operator=0, Delay=1000
EventTableTriggerLogic 8852: layoutX=96, layoutY=16, Operand1=cellC_pallet_holder 7125, Operand2=cellC_pallet_stopper 7126, Operator=0, Delay=1000
EventTableTriggerLogic 8853: layoutX=142, layoutY=32, Operand1=NOT 7128, Operand2=cellC_pallet_stopper 7127, Operator=0, Delay=1000
EventTableTriggerLogic 8854: layoutX=51, layoutY=46, Operand1=NOT 7130, Operand2=NOT 7132, Operator=0, Delay=1000
EventTableTriggerLogic 8855: layoutX=107, layoutY=60, Operand1=cellC_pallet_holder 7134, Operand2=NOT 7135, Operator=0, Delay=1000
EventTableTriggerIO 8856: IOValue=[1], IRC5Controller=? -1, Operator=0, SignalSource=ALab_CellC_v1.0_4 5362
EventTableTriggerLogic 8857: layoutX=184, layoutY=128, Operand1=AND 6402, Operand2=AND 6408, Operator=0, Delay=1000
EventTableTriggerLogic 8858: layoutX=231, layoutY=144, Operand1=AND 6416, Operand2=pallet1 6426, Operator=0, Delay=1000
EventTableTriggerLogic 8859: layoutX=251, layoutY=143, Operand1=AND 8115, Operand2=pallet3.1 8114, Operator=0, Delay=1000
EventTableTriggerLogic 8860: layoutX=62, layoutY=38, Operand1=pallet2 8126, Operand2=cellC_slider_horizontal_move 8125, Operator=0, Delay=1000
EventTableTriggerLogic 8861: layoutX=133, layoutY=37, Operand1=pallet3 6451, Operand2=pose6 6452, Operator=0, Delay=1000
EventTableTriggerLogic 8862: layoutX=61, layoutY=50, Operand1=pallet3.2 6456, Operand2=pose3 6457, Operator=0, Delay=1000
EventTableTriggerLogic 8863: layoutX=131, layoutY=52, Operand1=pickpallet1 6461, Operand2=pose7 6462, Operator=0, Delay=1000
EventTableTriggerLogic 8864: layoutX=8, layoutY=16, Operand1=pickpallet2 6466, Operand2=pose13 6467, Operator=0, Delay=1000
EventTableTriggerLogic 8865: layoutX=232, layoutY=117, Operand1=AND 6471, Operand2=pallet4 6481, Operator=0, Delay=1000
EventTableTriggerLogic 8866: layoutX=237, layoutY=122, Operand1=AND 6485, Operand2=conv2_buffer_stopper 6492, Operator=0, Delay=1000
EventTableTriggerLogic 8867: layoutX=240, layoutY=90, Operand1=AND 6496, Operand2=AND 6500, Operator=0, Delay=1000
EventTableTriggerLogic 8868: layoutX=80, layoutY=49, Operand1=pallet5.1 6513, Operand2=conv2_outer_lifter 6514, Operator=0, Delay=1000
EventTableTriggerIO 8869: IOValue=[1], IRC5Controller=? -1, Operator=0, SignalSource=LCFA_profile 1
EventTableTriggerIO 8870: IOValue=[1], IRC5Controller=? -1, Operator=0, SignalSource=LCFA_profile 1
EventTableTriggerIO 8871: IOValue=[1], IRC5Controller=? -1, Operator=0, SignalSource=LCFA_profile 1
EventTableTriggerIO 8872: IOValue=[1], IRC5Controller=? -1, Operator=0, SignalSource=LCFA_profile 1
EventTableTriggerIO 8873: IOValue=[1], IRC5Controller=? -1, Operator=0, SignalSource=LCFA_profile 1
EventTableTriggerIO 8874: IOValue=[1], IRC5Controller=? -1, Operator=0, SignalSource=LCFA_profile 1
EventTableTriggerIO 8875: IOValue=[1], IRC5Controller=? -1, Operator=0, SignalSource=LCFA_profile 1
EventTableTriggerIO 8876: IOValue=[1], IRC5Controller=? -1, Operator=0, SignalSource=LCFA_profile 1
EventTableTriggerIO 8877: IOValue=[1], IRC5Controller=? -1, Operator=0, SignalSource=LCFA_profile 1
EventTableTriggerIO 8878: IOValue=[1], IRC5Controller=? -1, Operator=0, SignalSource=LCFA_profile 1
EventTableTriggerIO 8879: IOValue=[0], IRC5Controller=? -1, Operator=0, SignalSource=ALab_CellC_v1.0_4 5362
EventTableTriggerIO 8880: IOValue=[1], IRC5Controller=? -1, Operator=0, SignalSource=ALab_CellC_v1.0_4 5362
EventTableTriggerIO 8881: IOValue=[0], IRC5Controller=? -1, Operator=0, SignalSource=ALab_CellC_v1.0_4 5362
EventTableTriggerIO 8882: IOValue=[1], IRC5Controller=? -1, Operator=0, SignalSource=ALab_CellC_v1.0_4 5362
EventTableTriggerIO 8883: IOValue=[1], IRC5Controller=? -1, Operator=0, SignalSource=ALab_CellC_v1.0_4 5362
EventTableTriggerIO 8884: IOValue=[0], IRC5Controller=? -1, Operator=0, SignalSource=ALab_CellC_v1.0_4 5362
EventTableTriggerIO 8885: IOValue=[0], IRC5Controller=? -1, Operator=0, SignalSource=ALab_CellC_v1.0_4 5362
EventTableTriggerIO 8886: IOValue=[1], IRC5Controller=? -1, Operator=0, SignalSource=ALab_CellC_v1.0_4 5362
EventTableTriggerIO 8887: IOValue=[1], IRC5Controller=? -1, Operator=0, SignalSource=ALab_CellC_v1.0_4 5362
EventTableTriggerIO 8888: IOValue=[0], IRC5Controller=? -1, Operator=0, SignalSource=ALab_CellC_v1.0_4 5362
EventTableTriggerIO 8889: IOValue=[1], IRC5Controller=? -1, Operator=0, SignalSource=ALab_CellC_v1.0_4 5362
EventTableTriggerIO 8890: IOValue=[0], IRC5Controller=? -1, Operator=0, SignalSource=ALab_CellC_v1.0_4 5362
EventTableTriggerIO 8891: IOValue=[0], IRC5Controller=? -1, Operator=0, SignalSource=ALab_CellC_v1.0_4 5362
EventTableTriggerIO 8892: IOValue=[1], IRC5Controller=? -1, Operator=0, SignalSource=ALab_CellC_v1.0_4 5362
EventTableTriggerIO 8893: IOValue=[1], IRC5Controller=? -1, Operator=0, SignalSource=ALab_CellC_v1.0_4 5362
EventTableTriggerIO 8894: IOValue=[0], IRC5Controller=? -1, Operator=0, SignalSource=ALab_CellC_v1.0_4 5362
EventTableTriggerIO 8895: IOValue=[0], IRC5Controller=? -1, Operator=0, SignalSource=ALab_CellC_v1.0_4 5362
EventTableTriggerIO 8896: IOValue=[1], IRC5Controller=? -1, Operator=0, SignalSource=ALab_CellC_v1.0_4 5362
EventTableTriggerIO 8897: IOValue=[1], IRC5Controller=? -1, Operator=0, SignalSource=ALab_CellC_v1.0_4 5362
EventTableTriggerIO 8898: IOValue=[0], IRC5Controller=? -1, Operator=0, SignalSource=ALab_CellC_v1.0_4 5362
EventTableTriggerIO 8899: IOValue=[1], IRC5Controller=? -1, Operator=0, SignalSource=LCFA_profile 1
EventTableTriggerIO 8900: IOValue=[1], IRC5Controller=? -1, Operator=0, SignalSource=LCFA_profile 1
EventTableTriggerIO 8901: IOValue=[1], IRC5Controller=? -1, Operator=0, SignalSource=LCFA_profile 1
EventTableTriggerIO 8902: IOValue=[1], IRC5Controller=? -1, Operator=0, SignalSource=LCFA_profile 1
EventTableTriggerIO 8903: IOValue=[1], IRC5Controller=? -1, Operator=0, SignalSource=ALab_CellC_v1.0_4 5362
EventTableTriggerIO 8904: IOValue=[0], IRC5Controller=? -1, Operator=0, SignalSource=ALab_CellC_v1.0_4 5362
EventTableTriggerIO 8905: IOValue=[1], IRC5Controller=? -1, Operator=0, SignalSource=LCFA_profile 1
EventTableTriggerIO 8906: IOValue=[1], IRC5Controller=? -1, Operator=0, SignalSource=LCFA_profile 1
EventTableTriggerIO 8907: IOValue=[1], IRC5Controller=? -1, Operator=0, SignalSource=LCFA_profile 1
EventTableTriggerIO 8908: IOValue=[1], IRC5Controller=? -1, Operator=0, SignalSource=LCFA_profile 1
EventTableTriggerIO 8909: IOValue=[1], IRC5Controller=? -1, Operator=0, SignalSource=ALab_CellC_v1.0_4 5362
EventTableTriggerIO 8910: IOValue=[0], IRC5Controller=? -1, Operator=0, SignalSource=ALab_CellC_v1.0_4 5362
EventTableTriggerIO 8911: IOValue=[1], IRC5Controller=? -1, Operator=0, SignalSource=ALab_CellC_v1.0_4 5362
EventTableTriggerIO 8912: IOValue=[0], IRC5Controller=? -1, Operator=0, SignalSource=ALab_CellC_v1.0_4 5362
EventTableTriggerIO 8913: IOValue=[0], IRC5Controller=? -1, Operator=0, SignalSource=ALab_CellC_v1.0_4 5362
EventTableTriggerIO 8914: IOValue=[1], IRC5Controller=? -1, Operator=0, SignalSource=ALab_CellC_v1.0_4 5362
EventTableTriggerIO 8915: IOValue=[1], IRC5Controller=? -1, Operator=0, SignalSource=ALab_CellC_v1.0_4 5362
EventTableTriggerIO 8916: IOValue=[0], IRC5Controller=? -1, Operator=0, SignalSource=ALab_CellC_v1.0_4 5362
EventTableTriggerIO 8917: IOValue=[1], IRC5Controller=? -1, Operator=0, SignalSource=LCFA_profile 1
EventTableTriggerIO 8918: IOValue=[1], IRC5Controller=? -1, Operator=0, SignalSource=LCFA_profile 1
EventTableTriggerIO 8919: IOValue=[1], IRC5Controller=? -1, Operator=0, SignalSource=LCFA_profile 1
EventTableTriggerLogic 8920: layoutX=150, layoutY=90, Operand1=AND 6770, Operand2=conv2_motor_s1 6766, Operator=0, Delay=1000
EventTableTriggerIO 8921: IOValue=[1], IRC5Controller=? -1, Operator=0, SignalSource=LCFA_profile 1
EventTableTriggerIO 8922: IOValue=[1], IRC5Controller=? -1, Operator=0, SignalSource=LCFA_profile 1
EventTableTriggerIO 8923: IOValue=[1], IRC5Controller=? -1, Operator=0, SignalSource=LCFA_profile 1
EventTableTriggerIO 8924: IOValue=[1], IRC5Controller=? -1, Operator=0, SignalSource=LCFA_profile 1
EventTableTriggerIO 8925: IOValue=[1], IRC5Controller=? -1, Operator=0, SignalSource=LCFA_profile 1
EventTableTriggerIO 8926: IOValue=[1], IRC5Controller=? -1, Operator=0, SignalSource=LCFA_profile 1
EventTableTriggerIO 8927: IOValue=[1], IRC5Controller=? -1, Operator=0, SignalSource=LCFA_profile 1
EventTableTriggerIO 8928: IOValue=[1], IRC5Controller=? -1, Operator=0, SignalSource=LCFA_profile 1
EventTableTriggerIO 8929: IOValue=[1], IRC5Controller=? -1, Operator=0, SignalSource=LCFA_profile 1
EventTableTriggerIO 8930: IOValue=[1], IRC5Controller=? -1, Operator=0, SignalSource=LCFA_profile 1
EventTableTriggerIO 8931: IOValue=[1], IRC5Controller=? -1, Operator=0, SignalSource=LCFA_profile 1
EventTableTriggerIO 8932: IOValue=[1], IRC5Controller=? -1, Operator=0, SignalSource=LCFA_profile 1
EventTableTriggerLogic 8933: layoutX=155, layoutY=137, Operand1=AND 6751, Operand2=NOT 6755, Operator=0, Delay=1000
EventTableTriggerIO 8934: IOValue=[1], IRC5Controller=? -1, Operator=0, SignalSource=LCFA_profile 1
EventTableTriggerIO 8935: IOValue=[1], IRC5Controller=? -1, Operator=0, SignalSource=LCFA_profile 1
EventTableTriggerLogic 8936: layoutX=48, layoutY=41, Operand1=pallet1.1 6778, Operand2=PalletIO00 6779, Operator=0, Delay=1000
EventTableTriggerIO 8937: IOValue=[1], IRC5Controller=? -1, Operator=0, SignalSource=LCFA_profile 1
EventTableTriggerIO 8938: IOValue=[1], IRC5Controller=? -1, Operator=0, SignalSource=ALab_CellC_v1.0_4 5362
EventTableTriggerIO 8939: IOValue=[0], IRC5Controller=? -1, Operator=0, SignalSource=ALab_CellC_v1.0_4 5362
EventTableTriggerLogic 8940: layoutX=103, layoutY=47, Operand1=NOT 8291, Operand2=pallet5 8290, Operator=0, Delay=1000
EventTableTriggerLogic 8941: layoutX=79, layoutY=37, Operand1=Pallet5.3 8029, Operand2=conv2_buffer_upper_vertical_move 8133, Operator=0, Delay=1000
EventTableTriggerLogic 8942: layoutX=40, layoutY=37, Operand1=Pallet5.4 8035, Operand2=conv2_buffer_lower_vertical_move 8036, Operator=0, Delay=1000
EventTableTriggerLogic 8943: layoutX=103, layoutY=47, Operand1=conv2_buffer_horizontal_move 8134, Operand2=Pallet5.7 8040, Operator=0, Delay=1000
EventTableTriggerLogic 8944: layoutX=54, layoutY=45, Operand1=NOT 8135, Operand2=Pallet5.6 8046, Operator=0, Delay=1000
EventTableTriggerLogic 8945: layoutX=108, layoutY=46, Operand1=NOT 8052, Operand2=Pallet5.5 8051, Operator=0, Delay=1000
EventTableTriggerIO 8946: IOValue=[1], IRC5Controller=? -1, Operator=0, SignalSource=LCFA_profile 1
EventTableTriggerIO 8947: IOValue=[1], IRC5Controller=? -1, Operator=0, SignalSource=LCFA_profile 1
EventTableTriggerIO 8948: IOValue=[1], IRC5Controller=? -1, Operator=0, SignalSource=LCFA_profile 1
EventTableTriggerIO 8949: IOValue=[1], IRC5Controller=? -1, Operator=0, SignalSource=LCFA_profile 1
EventTableTriggerIO 8950: IOValue=[1], IRC5Controller=? -1, Operator=0, SignalSource=LCFA_profile 1
EventTableTriggerIO 8951: IOValue=[1], IRC5Controller=? -1, Operator=0, SignalSource=LCFA_profile 1
EventTableTriggerIO 8952: IOValue=[1], IRC5Controller=? -1, Operator=0, SignalSource=LCFA_profile 1
EventTableTriggerIO 8953: IOValue=[1], IRC5Controller=? -1, Operator=0, SignalSource=LCFA_profile 1
EventTableTriggerIO 8954: IOValue=[1], IRC5Controller=? -1, Operator=0, SignalSource=LCFA_profile 1
EventTableTriggerIO 8955: IOValue=[1], IRC5Controller=? -1, Operator=0, SignalSource=LCFA_profile 1
EventTableTriggerIO 8956: IOValue=[1], IRC5Controller=? -1, Operator=0, SignalSource=LCFA_profile 1
EventTableTriggerIO 8957: IOValue=[1], IRC5Controller=? -1, Operator=0, SignalSource=LCFA_profile 1
EventTableTriggerIO 8958: IOValue=[1], IRC5Controller=? -1, Operator=0, SignalSource=LCFA_profile 1
EventTableTriggerIO 8959: IOValue=[1], IRC5Controller=? -1, Operator=0, SignalSource=LCFA_profile 1
EventTableTriggerIO 8960: IOValue=[1], IRC5Controller=? -1, Operator=0, SignalSource=LCFA_profile 1
EventTableTriggerIO 8961: IOValue=[1], IRC5Controller=? -1, Operator=0, SignalSource=LCFA_profile 1
EventTableTriggerIO 8962: IOValue=[1], IRC5Controller=? -1, Operator=0, SignalSource=LCFA_profile 1
EventTableTriggerLogic 8963: layoutX=99, layoutY=32, Operand1=Pallet2.1 8141, Operand2=NOT 8139, Operator=0, Delay=1000
EventTableTriggerLogic 8964: layoutX=181, layoutY=52, Operand1=conv1_buffer_upper_go_down 8146, Operand2=Pallet2.2 8145, Operator=0, Delay=1000
EventTableTriggerLogic 8965: layoutX=48, layoutY=51, Operand1=Pallet2.3 8150, Operand2=conv1_buffer_lower_go_up 8151, Operator=0, Delay=1000
EventTableTriggerLogic 8966: layoutX=67, layoutY=33, Operand1=pallet2 8155, Operand2=NOT 8156, Operator=0, Delay=1000
EventTableTriggerLogic 8967: layoutX=102, layoutY=29, Operand1=Pallet2.4 8161, Operand2=NOT 8162, Operator=0, Delay=1000
EventTableTriggerLogic 8968: layoutX=102, layoutY=23, Operand1=Pallet2.5 8167, Operand2=NOT 8168, Operator=0, Delay=1000
EventTableTriggerIO 8969: IOValue=[1], IRC5Controller=? -1, Operator=0, SignalSource=LCFA_profile 1
EventTableTriggerIO 8970: IOValue=[1], IRC5Controller=? -1, Operator=0, SignalSource=LCFA_profile 1
EventTableTriggerIO 8971: IOValue=[1], IRC5Controller=? -1, Operator=0, SignalSource=LCFA_profile 1
EventTableTriggerIO 8972: IOValue=[1], IRC5Controller=? -1, Operator=0, SignalSource=LCFA_profile 1
EventTableTriggerIO 8973: IOValue=[1], IRC5Controller=? -1, Operator=0, SignalSource=LCFA_profile 1
EventTableTriggerIO 8974: IOValue=[1], IRC5Controller=? -1, Operator=0, SignalSource=LCFA_profile 1
EventTableTriggerIO 8975: IOValue=[1], IRC5Controller=? -1, Operator=0, SignalSource=LCFA_profile 1
EventTableTriggerIO 8976: IOValue=[1], IRC5Controller=? -1, Operator=0, SignalSource=LCFA_profile 1
EventTableTriggerIO 8977: IOValue=[1], IRC5Controller=? -1, Operator=0, SignalSource=LCFA_profile 1
EventTableTriggerIO 8978: IOValue=[1], IRC5Controller=? -1, Operator=0, SignalSource=LCFA_profile 1
EventTableTriggerIO 8979: IOValue=[1], IRC5Controller=? -1, Operator=0, SignalSource=LCFA_profile 1
EventTableTriggerIO 8980: IOValue=[1], IRC5Controller=? -1, Operator=0, SignalSource=LCFA_profile 1
EventTableTriggerIO 8981: IOValue=[1], IRC5Controller=? -1, Operator=0, SignalSource=LCFA_profile 1
EventTableTriggerLogic 8982: layoutX=49, layoutY=26, Operand1=Pallet2.6 8213, Operand2=conv1_buffer_horizontal_open 8214, Operator=0, Delay=1000
EventTableTriggerIO 8983: IOValue=[1], IRC5Controller=? -1, Operator=0, SignalSource=LCFA_profile 1
EventTableTriggerIO 8984: IOValue=[1], IRC5Controller=? -1, Operator=0, SignalSource=LCFA_profile 1
EventTableTriggerIO 8985: IOValue=[1], IRC5Controller=? -1, Operator=0, SignalSource=LCFA_profile 1
EventTableTriggerIO 8986: IOValue=[1], IRC5Controller=? -1, Operator=0, SignalSource=LCFA_profile 1
EventTableTriggerIO 8987: IOValue=[1], IRC5Controller=? -1, Operator=0, SignalSource=LCFA_profile 1
EventTableTriggerIO 8988: IOValue=[1], IRC5Controller=? -1, Operator=0, SignalSource=ALab_CellC_v1.0_4 5362
EventTableTriggerIO 8989: IOValue=[0], IRC5Controller=? -1, Operator=0, SignalSource=ALab_CellC_v1.0_4 5362
EventTableTriggerIO 8990: IOValue=[1], IRC5Controller=? -1, Operator=0, SignalSource=ALab_CellC_v1.0_4 5362
EventTableTriggerIO 8991: IOValue=[0], IRC5Controller=? -1, Operator=0, SignalSource=ALab_CellC_v1.0_4 5362
EventTableTriggerIO 8992: IOValue=[1], IRC5Controller=? -1, Operator=0, SignalSource=ALab_CellC_v1.0_4 5362
EventTableTriggerIO 8993: IOValue=[0], IRC5Controller=? -1, Operator=0, SignalSource=ALab_CellC_v1.0_4 5362
EventTableTriggerIO 8994: IOValue=[0], IRC5Controller=? -1, Operator=0, SignalSource=ALab_CellC_v1.0_4 5362
EventTableTriggerIO 8995: IOValue=[1], IRC5Controller=? -1, Operator=0, SignalSource=ALab_CellC_v1.0_4 5362
EventTableTriggerIO 8996: IOValue=[0], IRC5Controller=? -1, Operator=0, SignalSource=ALab_CellC_v1.0_4 5362
EventTableTriggerIO 8997: IOValue=[1], IRC5Controller=? -1, Operator=0, SignalSource=ALab_CellC_v1.0_4 5362
EventTableTriggerIO 8998: IOValue=[1], IRC5Controller=? -1, Operator=0, SignalSource=ALab_CellC_v1.0_4 5362
EventTableTriggerIO 8999: IOValue=[0], IRC5Controller=? -1, Operator=0, SignalSource=ALab_CellC_v1.0_4 5362
EventTableTriggerIO 9000: IOValue=[0], IRC5Controller=? -1, Operator=0, SignalSource=ALab_CellC_v1.0_4 5362
EventTableTriggerIO 9001: IOValue=[1], IRC5Controller=? -1, Operator=0, SignalSource=ALab_CellC_v1.0_4 5362
EventTableTriggerIO 9002: IOValue=[1], IRC5Controller=? -1, Operator=0, SignalSource=ALab_CellC_v1.0_4 5362
EventTableTriggerIO 9003: IOValue=[0], IRC5Controller=? -1, Operator=0, SignalSource=ALab_CellC_v1.0_4 5362
EventTableTriggerIO 9004: IOValue=[0], IRC5Controller=? -1, Operator=0, SignalSource=ALab_CellC_v1.0_4 5362
EventTableTriggerIO 9005: IOValue=[1], IRC5Controller=? -1, Operator=0, SignalSource=ALab_CellC_v1.0_4 5362
EventTableTriggerIO 9006: IOValue=[1], IRC5Controller=? -1, Operator=0, SignalSource=ALab_CellC_v1.0_4 5362
EventTableTriggerIO 9007: IOValue=[0], IRC5Controller=? -1, Operator=0, SignalSource=ALab_CellC_v1.0_4 5362
EventTableTriggerIO 9008: IOValue=[1], IRC5Controller=? -1, Operator=0, SignalSource=LCFA_profile 1
EventTableTriggerIO 9009: IOValue=[1], IRC5Controller=? -1, Operator=0, SignalSource=LCFA_profile 1
EventTableTriggerIO 9010: IOValue=[1], IRC5Controller=? -1, Operator=0, SignalSource=ALab_CellC_v1.0_4 5362
EventTableTriggerIO 9011: IOValue=[0], IRC5Controller=? -1, Operator=0, SignalSource=ALab_CellC_v1.0_4 5362
EventTableTriggerIO 9012: IOValue=[1], IRC5Controller=? -1, Operator=0, SignalSource=ALab_CellC_v1.0_4 5362
EventTableTriggerIO 9013: IOValue=[0], IRC5Controller=? -1, Operator=0, SignalSource=ALab_CellC_v1.0_4 5362
EventTableTriggerLogic 9107: layoutX=167, layoutY=76, Operand1=AND 4076, Operand2=AND 4081, Operator=0, Delay=1000
EventTableTriggerLogic 9108: layoutX=194, layoutY=70, Operand1=AND 4088, Operand2=AND 4093, Operator=0, Delay=1000
EventTableTriggerLogic 9109: layoutX=181, layoutY=88, Operand1=AND 4100, Operand2=AND 4105, Operator=0, Delay=1000
EventTableTriggerLogic 9110: layoutX=165, layoutY=70, Operand1=AND 4112, Operand2=AND 4117, Operator=0, Delay=1000
EventTableTriggerLogic 9111: layoutX=217, layoutY=77, Operand1=AND 4123, Operand2=AND 4127, Operator=0, Delay=1000
EventTableTriggerLogic 9112: layoutX=168, layoutY=84, Operand1=AND 4135, Operand2=AND 4139, Operator=0, Delay=1000
EventTableTriggerLogic 9113: layoutX=219, layoutY=73, Operand1=AND 4146, Operand2=AND 4150, Operator=0, Delay=1000
EventTableTriggerLogic 9114: layoutX=203, layoutY=67, Operand1=AND 4157, Operand2=AND 4161, Operator=0, Delay=1000
EventTableTriggerLogic 9115: layoutX=220, layoutY=69, Operand1=AND 4167, Operand2=AND 4171, Operator=0, Delay=1000
EventTableTriggerLogic 9116: layoutX=243, layoutY=55, Operand1=AND 4179, Operand2=AND 4183, Operator=0, Delay=1000
EventTableTriggerLogic 9117: layoutX=204, layoutY=112, Operand1=AND 4190, Operand2=AND 4194, Operator=0, Delay=1000
EventTableTriggerLogic 9118: layoutX=245, layoutY=97, Operand1=AND 4201, Operand2=AND 4205, Operator=0, Delay=1000
EventTableTriggerLogic 9119: layoutX=234, layoutY=61, Operand1=AND 4211, Operand2=AND 4214, Operator=0, Delay=1000
EventTableTriggerLogic 9120: layoutX=192, layoutY=87, Operand1=AND 4222, Operand2=AND 4225, Operator=0, Delay=1000
EventTableTriggerLogic 9121: layoutX=212, layoutY=64, Operand1=AND 4232, Operand2=AND 4235, Operator=0, Delay=1000
EventTableTriggerLogic 9122: layoutX=160, layoutY=73, Operand1=AND 4242, Operand2=AND 4245, Operator=0, Delay=1000
EventTableTriggerLogic 9123: layoutX=153, layoutY=73, Operand1=AND 4264, Operand2=NOT 4269, Operator=0, Delay=1000
EventTableTriggerLogic 9124: layoutX=133, layoutY=81, Operand1=AND 4274, Operand2=conv1_buffer_upper_go_down 6332, Operator=0, Delay=1000
EventTableTriggerLogic 9125: layoutX=184, layoutY=91, Operand1=AND 4283, Operand2=NOT 4287, Operator=0, Delay=1000
EventTableTriggerLogic 9126: layoutX=211, layoutY=90, Operand1=AND 4292, Operand2=conv1_buffer_upper_go_down 6282, Operator=0, Delay=1000
EventTableTriggerLogic 9127: layoutX=226, layoutY=110, Operand1=AND 4300, Operand2=NOT 4304, Operator=0, Delay=1000
EventTableTriggerLogic 9128: layoutX=164, layoutY=68, Operand1=AND 4309, Operand2=conv1_buffer_upper_go_down 6288, Operator=0, Delay=1000
EventTableTriggerLogic 9129: layoutX=161, layoutY=63, Operand1=AND 4317, Operand2=NOT 4320, Operator=0, Delay=1000
EventTableTriggerLogic 9130: layoutX=174, layoutY=87, Operand1=AND 4325, Operand2=conv1_buffer_upper_go_down 6294, Operator=0, Delay=1000
EventTableTriggerLogic 9131: layoutX=148, layoutY=98, Operand1=AND 4332, Operand2=NOT 4337, Operator=0, Delay=1000
EventTableTriggerLogic 9132: layoutX=206, layoutY=74, Operand1=AND 4342, Operand2=conv2_buffer_upper_vertical_move 6300, Operator=0, Delay=1000
EventTableTriggerLogic 9133: layoutX=195, layoutY=82, Operand1=AND 4351, Operand2=NOT 4355, Operator=0, Delay=1000
EventTableTriggerLogic 9134: layoutX=193, layoutY=94, Operand1=AND 4360, Operand2=conv2_buffer_upper_vertical_move 6306, Operator=0, Delay=1000
EventTableTriggerLogic 9135: layoutX=210, layoutY=27, Operand1=conv2_buffer_horizontal_move 6309, Operand2=AND 4369, Operator=0, Delay=1000
EventTableTriggerLogic 9136: layoutX=233, layoutY=95, Operand1=AND 4377, Operand2=conv2_buffer_upper_vertical_move 6312, Operator=0, Delay=1000
EventTableTriggerLogic 9137: layoutX=102, layoutY=69, Operand1=AND 4385, Operand2=NOT 4388, Operator=0, Delay=1000
EventTableTriggerLogic 9138: layoutX=97, layoutY=92, Operand1=AND 4393, Operand2=conv2_buffer_upper_vertical_move 6318, Operator=0, Delay=1000
EventTableTriggerLogic 9139: layoutX=96, layoutY=16, Operand1=cellC_pallet_holder 7125, Operand2=cellC_pallet_stopper 7126, Operator=0, Delay=1000
EventTableTriggerLogic 9140: layoutX=142, layoutY=32, Operand1=NOT 7128, Operand2=cellC_pallet_stopper 7127, Operator=0, Delay=1000
EventTableTriggerLogic 9141: layoutX=51, layoutY=46, Operand1=NOT 7130, Operand2=NOT 7132, Operator=0, Delay=1000
EventTableTriggerLogic 9142: layoutX=107, layoutY=60, Operand1=cellC_pallet_holder 7134, Operand2=NOT 7135, Operator=0, Delay=1000
EventTableTriggerIO 9143: IOValue=[1], IRC5Controller=? -1, Operator=0, SignalSource=ALab_CellC_v1.0_4 5362
EventTableTriggerLogic 9144: layoutX=184, layoutY=128, Operand1=AND 6402, Operand2=AND 6408, Operator=0, Delay=1000
EventTableTriggerLogic 9145: layoutX=231, layoutY=144, Operand1=AND 6416, Operand2=pallet1 6426, Operator=0, Delay=1000
EventTableTriggerLogic 9146: layoutX=251, layoutY=143, Operand1=AND 8115, Operand2=pallet3.1 8114, Operator=0, Delay=1000
EventTableTriggerLogic 9147: layoutX=62, layoutY=38, Operand1=pallet2 8126, Operand2=cellC_slider_horizontal_move 8125, Operator=0, Delay=1000
EventTableTriggerLogic 9148: layoutX=133, layoutY=37, Operand1=pallet3 6451, Operand2=pose6 6452, Operator=0, Delay=1000
EventTableTriggerLogic 9149: layoutX=61, layoutY=50, Operand1=pallet3.2 6456, Operand2=pose3 6457, Operator=0, Delay=1000
EventTableTriggerLogic 9150: layoutX=131, layoutY=52, Operand1=pickpallet1 6461, Operand2=pose7 6462, Operator=0, Delay=1000
EventTableTriggerLogic 9151: layoutX=8, layoutY=16, Operand1=pickpallet2 6466, Operand2=pose13 6467, Operator=0, Delay=1000
EventTableTriggerLogic 9152: layoutX=232, layoutY=117, Operand1=AND 6471, Operand2=pallet4 6481, Operator=0, Delay=1000
EventTableTriggerLogic 9153: layoutX=237, layoutY=122, Operand1=AND 6485, Operand2=conv2_buffer_stopper 6492, Operator=0, Delay=1000
EventTableTriggerLogic 9154: layoutX=240, layoutY=90, Operand1=AND 6496, Operand2=AND 6500, Operator=0, Delay=1000
EventTableTriggerLogic 9155: layoutX=80, layoutY=49, Operand1=pallet5.1 6513, Operand2=conv2_outer_lifter 6514, Operator=0, Delay=1000
EventTableTriggerIO 9156: IOValue=[1], IRC5Controller=? -1, Operator=0, SignalSource=LCFA_profile 1
EventTableTriggerIO 9157: IOValue=[1], IRC5Controller=? -1, Operator=0, SignalSource=LCFA_profile 1
EventTableTriggerIO 9158: IOValue=[1], IRC5Controller=? -1, Operator=0, SignalSource=LCFA_profile 1
EventTableTriggerIO 9159: IOValue=[1], IRC5Controller=? -1, Operator=0, SignalSource=LCFA_profile 1
EventTableTriggerIO 9160: IOValue=[1], IRC5Controller=? -1, Operator=0, SignalSource=LCFA_profile 1
EventTableTriggerIO 9161: IOValue=[1], IRC5Controller=? -1, Operator=0, SignalSource=LCFA_profile 1
EventTableTriggerIO 9162: IOValue=[1], IRC5Controller=? -1, Operator=0, SignalSource=LCFA_profile 1
EventTableTriggerIO 9163: IOValue=[1], IRC5Controller=? -1, Operator=0, SignalSource=LCFA_profile 1
EventTableTriggerIO 9164: IOValue=[1], IRC5Controller=? -1, Operator=0, SignalSource=LCFA_profile 1
EventTableTriggerIO 9165: IOValue=[1], IRC5Controller=? -1, Operator=0, SignalSource=LCFA_profile 1
EventTableTriggerIO 9166: IOValue=[0], IRC5Controller=? -1, Operator=0, SignalSource=ALab_CellC_v1.0_4 5362
EventTableTriggerIO 9167: IOValue=[1], IRC5Controller=? -1, Operator=0, SignalSource=ALab_CellC_v1.0_4 5362
EventTableTriggerIO 9168: IOValue=[0], IRC5Controller=? -1, Operator=0, SignalSource=ALab_CellC_v1.0_4 5362
EventTableTriggerIO 9169: IOValue=[1], IRC5Controller=? -1, Operator=0, SignalSource=ALab_CellC_v1.0_4 5362
EventTableTriggerIO 9170: IOValue=[1], IRC5Controller=? -1, Operator=0, SignalSource=ALab_CellC_v1.0_4 5362
EventTableTriggerIO 9171: IOValue=[0], IRC5Controller=? -1, Operator=0, SignalSource=ALab_CellC_v1.0_4 5362
EventTableTriggerIO 9172: IOValue=[0], IRC5Controller=? -1, Operator=0, SignalSource=ALab_CellC_v1.0_4 5362
EventTableTriggerIO 9173: IOValue=[1], IRC5Controller=? -1, Operator=0, SignalSource=ALab_CellC_v1.0_4 5362
EventTableTriggerIO 9174: IOValue=[1], IRC5Controller=? -1, Operator=0, SignalSource=ALab_CellC_v1.0_4 5362
EventTableTriggerIO 9175: IOValue=[0], IRC5Controller=? -1, Operator=0, SignalSource=ALab_CellC_v1.0_4 5362
EventTableTriggerIO 9176: IOValue=[1], IRC5Controller=? -1, Operator=0, SignalSource=ALab_CellC_v1.0_4 5362
EventTableTriggerIO 9177: IOValue=[0], IRC5Controller=? -1, Operator=0, SignalSource=ALab_CellC_v1.0_4 5362
EventTableTriggerIO 9178: IOValue=[0], IRC5Controller=? -1, Operator=0, SignalSource=ALab_CellC_v1.0_4 5362
EventTableTriggerIO 9179: IOValue=[1], IRC5Controller=? -1, Operator=0, SignalSource=ALab_CellC_v1.0_4 5362
EventTableTriggerIO 9180: IOValue=[1], IRC5Controller=? -1, Operator=0, SignalSource=ALab_CellC_v1.0_4 5362
EventTableTriggerIO 9181: IOValue=[0], IRC5Controller=? -1, Operator=0, SignalSource=ALab_CellC_v1.0_4 5362
EventTableTriggerIO 9182: IOValue=[0], IRC5Controller=? -1, Operator=0, SignalSource=ALab_CellC_v1.0_4 5362
EventTableTriggerIO 9183: IOValue=[1], IRC5Controller=? -1, Operator=0, SignalSource=ALab_CellC_v1.0_4 5362
EventTableTriggerIO 9184: IOValue=[1], IRC5Controller=? -1, Operator=0, SignalSource=ALab_CellC_v1.0_4 5362
EventTableTriggerIO 9185: IOValue=[0], IRC5Controller=? -1, Operator=0, SignalSource=ALab_CellC_v1.0_4 5362
EventTableTriggerIO 9186: IOValue=[1], IRC5Controller=? -1, Operator=0, SignalSource=LCFA_profile 1
EventTableTriggerIO 9187: IOValue=[1], IRC5Controller=? -1, Operator=0, SignalSource=LCFA_profile 1
EventTableTriggerIO 9188: IOValue=[1], IRC5Controller=? -1, Operator=0, SignalSource=LCFA_profile 1
EventTableTriggerIO 9189: IOValue=[1], IRC5Controller=? -1, Operator=0, SignalSource=LCFA_profile 1
EventTableTriggerIO 9190: IOValue=[1], IRC5Controller=? -1, Operator=0, SignalSource=ALab_CellC_v1.0_4 5362
EventTableTriggerIO 9191: IOValue=[0], IRC5Controller=? -1, Operator=0, SignalSource=ALab_CellC_v1.0_4 5362
EventTableTriggerIO 9192: IOValue=[1], IRC5Controller=? -1, Operator=0, SignalSource=LCFA_profile 1
EventTableTriggerIO 9193: IOValue=[1], IRC5Controller=? -1, Operator=0, SignalSource=LCFA_profile 1
EventTableTriggerIO 9194: IOValue=[1], IRC5Controller=? -1, Operator=0, SignalSource=LCFA_profile 1
EventTableTriggerIO 9195: IOValue=[1], IRC5Controller=? -1, Operator=0, SignalSource=LCFA_profile 1
EventTableTriggerIO 9196: IOValue=[1], IRC5Controller=? -1, Operator=0, SignalSource=ALab_CellC_v1.0_4 5362
EventTableTriggerIO 9197: IOValue=[0], IRC5Controller=? -1, Operator=0, SignalSource=ALab_CellC_v1.0_4 5362
EventTableTriggerIO 9198: IOValue=[1], IRC5Controller=? -1, Operator=0, SignalSource=ALab_CellC_v1.0_4 5362
EventTableTriggerIO 9199: IOValue=[0], IRC5Controller=? -1, Operator=0, SignalSource=ALab_CellC_v1.0_4 5362
EventTableTriggerIO 9200: IOValue=[0], IRC5Controller=? -1, Operator=0, SignalSource=ALab_CellC_v1.0_4 5362
EventTableTriggerIO 9201: IOValue=[1], IRC5Controller=? -1, Operator=0, SignalSource=ALab_CellC_v1.0_4 5362
EventTableTriggerIO 9202: IOValue=[1], IRC5Controller=? -1, Operator=0, SignalSource=ALab_CellC_v1.0_4 5362
EventTableTriggerIO 9203: IOValue=[0], IRC5Controller=? -1, Operator=0, SignalSource=ALab_CellC_v1.0_4 5362
EventTableTriggerIO 9204: IOValue=[1], IRC5Controller=? -1, Operator=0, SignalSource=LCFA_profile 1
EventTableTriggerIO 9205: IOValue=[1], IRC5Controller=? -1, Operator=0, SignalSource=LCFA_profile 1
EventTableTriggerIO 9206: IOValue=[1], IRC5Controller=? -1, Operator=0, SignalSource=LCFA_profile 1
EventTableTriggerLogic 9207: layoutX=150, layoutY=90, Operand1=AND 6770, Operand2=conv2_motor_s1 6766, Operator=0, Delay=1000
EventTableTriggerIO 9208: IOValue=[1], IRC5Controller=? -1, Operator=0, SignalSource=LCFA_profile 1
EventTableTriggerIO 9209: IOValue=[1], IRC5Controller=? -1, Operator=0, SignalSource=LCFA_profile 1
EventTableTriggerIO 9210: IOValue=[1], IRC5Controller=? -1, Operator=0, SignalSource=LCFA_profile 1
EventTableTriggerIO 9211: IOValue=[1], IRC5Controller=? -1, Operator=0, SignalSource=LCFA_profile 1
EventTableTriggerIO 9212: IOValue=[1], IRC5Controller=? -1, Operator=0, SignalSource=LCFA_profile 1
EventTableTriggerIO 9213: IOValue=[1], IRC5Controller=? -1, Operator=0, SignalSource=LCFA_profile 1
EventTableTriggerIO 9214: IOValue=[1], IRC5Controller=? -1, Operator=0, SignalSource=LCFA_profile 1
EventTableTriggerIO 9215: IOValue=[1], IRC5Controller=? -1, Operator=0, SignalSource=LCFA_profile 1
EventTableTriggerIO 9216: IOValue=[1], IRC5Controller=? -1, Operator=0, SignalSource=LCFA_profile 1
EventTableTriggerIO 9217: IOValue=[1], IRC5Controller=? -1, Operator=0, SignalSource=LCFA_profile 1
EventTableTriggerIO 9218: IOValue=[1], IRC5Controller=? -1, Operator=0, SignalSource=LCFA_profile 1
EventTableTriggerIO 9219: IOValue=[1], IRC5Controller=? -1, Operator=0, SignalSource=LCFA_profile 1
EventTableTriggerLogic 9220: layoutX=155, layoutY=137, Operand1=AND 6751, Operand2=NOT 6755, Operator=0, Delay=1000
EventTableTriggerIO 9221: IOValue=[1], IRC5Controller=? -1, Operator=0, SignalSource=LCFA_profile 1
EventTableTriggerIO 9222: IOValue=[1], IRC5Controller=? -1, Operator=0, SignalSource=LCFA_profile 1
EventTableTriggerLogic 9223: layoutX=48, layoutY=41, Operand1=pallet1.1 6778, Operand2=PalletIO00 6779, Operator=0, Delay=1000
EventTableTriggerIO 9224: IOValue=[1], IRC5Controller=? -1, Operator=0, SignalSource=LCFA_profile 1
EventTableTriggerIO 9225: IOValue=[1], IRC5Controller=? -1, Operator=0, SignalSource=ALab_CellC_v1.0_4 5362
EventTableTriggerIO 9226: IOValue=[0], IRC5Controller=? -1, Operator=0, SignalSource=ALab_CellC_v1.0_4 5362
EventTableTriggerLogic 9227: layoutX=103, layoutY=47, Operand1=NOT 8291, Operand2=pallet5 8290, Operator=0, Delay=1000
EventTableTriggerLogic 9228: layoutX=79, layoutY=37, Operand1=Pallet5.3 8029, Operand2=conv2_buffer_upper_vertical_move 8133, Operator=0, Delay=1000
EventTableTriggerLogic 9229: layoutX=40, layoutY=37, Operand1=Pallet5.4 8035, Operand2=conv2_buffer_lower_vertical_move 8036, Operator=0, Delay=1000
EventTableTriggerLogic 9230: layoutX=103, layoutY=47, Operand1=conv2_buffer_horizontal_move 8134, Operand2=Pallet5.7 8040, Operator=0, Delay=1000
EventTableTriggerLogic 9231: layoutX=54, layoutY=45, Operand1=NOT 8135, Operand2=Pallet5.6 8046, Operator=0, Delay=1000
EventTableTriggerLogic 9232: layoutX=108, layoutY=46, Operand1=NOT 8052, Operand2=Pallet5.5 8051, Operator=0, Delay=1000
EventTableTriggerIO 9233: IOValue=[1], IRC5Controller=? -1, Operator=0, SignalSource=LCFA_profile 1
EventTableTriggerIO 9234: IOValue=[1], IRC5Controller=? -1, Operator=0, SignalSource=LCFA_profile 1
EventTableTriggerIO 9235: IOValue=[1], IRC5Controller=? -1, Operator=0, SignalSource=LCFA_profile 1
EventTableTriggerIO 9236: IOValue=[1], IRC5Controller=? -1, Operator=0, SignalSource=LCFA_profile 1
EventTableTriggerIO 9237: IOValue=[1], IRC5Controller=? -1, Operator=0, SignalSource=LCFA_profile 1
EventTableTriggerIO 9238: IOValue=[1], IRC5Controller=? -1, Operator=0, SignalSource=LCFA_profile 1
EventTableTriggerIO 9239: IOValue=[1], IRC5Controller=? -1, Operator=0, SignalSource=LCFA_profile 1
EventTableTriggerIO 9240: IOValue=[1], IRC5Controller=? -1, Operator=0, SignalSource=LCFA_profile 1
EventTableTriggerIO 9241: IOValue=[1], IRC5Controller=? -1, Operator=0, SignalSource=LCFA_profile 1
EventTableTriggerIO 9242: IOValue=[1], IRC5Controller=? -1, Operator=0, SignalSource=LCFA_profile 1
EventTableTriggerIO 9243: IOValue=[1], IRC5Controller=? -1, Operator=0, SignalSource=LCFA_profile 1
EventTableTriggerIO 9244: IOValue=[1], IRC5Controller=? -1, Operator=0, SignalSource=LCFA_profile 1
EventTableTriggerIO 9245: IOValue=[1], IRC5Controller=? -1, Operator=0, SignalSource=LCFA_profile 1
EventTableTriggerIO 9246: IOValue=[1], IRC5Controller=? -1, Operator=0, SignalSource=LCFA_profile 1
EventTableTriggerIO 9247: IOValue=[1], IRC5Controller=? -1, Operator=0, SignalSource=LCFA_profile 1
EventTableTriggerIO 9248: IOValue=[1], IRC5Controller=? -1, Operator=0, SignalSource=LCFA_profile 1
EventTableTriggerIO 9249: IOValue=[1], IRC5Controller=? -1, Operator=0, SignalSource=LCFA_profile 1
EventTableTriggerLogic 9250: layoutX=99, layoutY=32, Operand1=Pallet2.1 8141, Operand2=NOT 8139, Operator=0, Delay=1000
EventTableTriggerLogic 9251: layoutX=181, layoutY=52, Operand1=conv1_buffer_upper_go_down 8146, Operand2=Pallet2.2 8145, Operator=0, Delay=1000
EventTableTriggerLogic 9252: layoutX=48, layoutY=51, Operand1=Pallet2.3 8150, Operand2=conv1_buffer_lower_go_up 8151, Operator=0, Delay=1000
EventTableTriggerLogic 9253: layoutX=67, layoutY=33, Operand1=pallet2 8155, Operand2=NOT 8156, Operator=0, Delay=1000
EventTableTriggerLogic 9254: layoutX=102, layoutY=29, Operand1=Pallet2.4 8161, Operand2=NOT 8162, Operator=0, Delay=1000
EventTableTriggerLogic 9255: layoutX=102, layoutY=23, Operand1=Pallet2.5 8167, Operand2=NOT 8168, Operator=0, Delay=1000
EventTableTriggerIO 9256: IOValue=[1], IRC5Controller=? -1, Operator=0, SignalSource=LCFA_profile 1
EventTableTriggerIO 9257: IOValue=[1], IRC5Controller=? -1, Operator=0, SignalSource=LCFA_profile 1
EventTableTriggerIO 9258: IOValue=[1], IRC5Controller=? -1, Operator=0, SignalSource=LCFA_profile 1
EventTableTriggerIO 9259: IOValue=[1], IRC5Controller=? -1, Operator=0, SignalSource=LCFA_profile 1
EventTableTriggerIO 9260: IOValue=[1], IRC5Controller=? -1, Operator=0, SignalSource=LCFA_profile 1
EventTableTriggerIO 9261: IOValue=[1], IRC5Controller=? -1, Operator=0, SignalSource=LCFA_profile 1
EventTableTriggerIO 9262: IOValue=[1], IRC5Controller=? -1, Operator=0, SignalSource=LCFA_profile 1
EventTableTriggerIO 9263: IOValue=[1], IRC5Controller=? -1, Operator=0, SignalSource=LCFA_profile 1
EventTableTriggerIO 9264: IOValue=[1], IRC5Controller=? -1, Operator=0, SignalSource=LCFA_profile 1
EventTableTriggerIO 9265: IOValue=[1], IRC5Controller=? -1, Operator=0, SignalSource=LCFA_profile 1
EventTableTriggerIO 9266: IOValue=[1], IRC5Controller=? -1, Operator=0, SignalSource=LCFA_profile 1
EventTableTriggerIO 9267: IOValue=[1], IRC5Controller=? -1, Operator=0, SignalSource=LCFA_profile 1
EventTableTriggerIO 9268: IOValue=[1], IRC5Controller=? -1, Operator=0, SignalSource=LCFA_profile 1
EventTableTriggerLogic 9269: layoutX=49, layoutY=26, Operand1=Pallet2.6 8213, Operand2=conv1_buffer_horizontal_open 8214, Operator=0, Delay=1000
EventTableTriggerIO 9270: IOValue=[1], IRC5Controller=? -1, Operator=0, SignalSource=LCFA_profile 1
EventTableTriggerIO 9271: IOValue=[1], IRC5Controller=? -1, Operator=0, SignalSource=LCFA_profile 1
EventTableTriggerIO 9272: IOValue=[1], IRC5Controller=? -1, Operator=0, SignalSource=LCFA_profile 1
EventTableTriggerIO 9273: IOValue=[1], IRC5Controller=? -1, Operator=0, SignalSource=LCFA_profile 1
EventTableTriggerIO 9274: IOValue=[1], IRC5Controller=? -1, Operator=0, SignalSource=LCFA_profile 1
EventTableTriggerIO 9275: IOValue=[1], IRC5Controller=? -1, Operator=0, SignalSource=ALab_CellC_v1.0_4 5362
EventTableTriggerIO 9276: IOValue=[0], IRC5Controller=? -1, Operator=0, SignalSource=ALab_CellC_v1.0_4 5362
EventTableTriggerIO 9277: IOValue=[1], IRC5Controller=? -1, Operator=0, SignalSource=ALab_CellC_v1.0_4 5362
EventTableTriggerIO 9278: IOValue=[0], IRC5Controller=? -1, Operator=0, SignalSource=ALab_CellC_v1.0_4 5362
EventTableTriggerIO 9279: IOValue=[1], IRC5Controller=? -1, Operator=0, SignalSource=ALab_CellC_v1.0_4 5362
EventTableTriggerIO 9280: IOValue=[0], IRC5Controller=? -1, Operator=0, SignalSource=ALab_CellC_v1.0_4 5362
EventTableTriggerIO 9281: IOValue=[0], IRC5Controller=? -1, Operator=0, SignalSource=ALab_CellC_v1.0_4 5362
EventTableTriggerIO 9282: IOValue=[1], IRC5Controller=? -1, Operator=0, SignalSource=ALab_CellC_v1.0_4 5362
EventTableTriggerIO 9283: IOValue=[0], IRC5Controller=? -1, Operator=0, SignalSource=ALab_CellC_v1.0_4 5362
EventTableTriggerIO 9284: IOValue=[1], IRC5Controller=? -1, Operator=0, SignalSource=ALab_CellC_v1.0_4 5362
EventTableTriggerIO 9285: IOValue=[1], IRC5Controller=? -1, Operator=0, SignalSource=ALab_CellC_v1.0_4 5362
EventTableTriggerIO 9286: IOValue=[0], IRC5Controller=? -1, Operator=0, SignalSource=ALab_CellC_v1.0_4 5362
EventTableTriggerIO 9287: IOValue=[0], IRC5Controller=? -1, Operator=0, SignalSource=ALab_CellC_v1.0_4 5362
EventTableTriggerIO 9288: IOValue=[1], IRC5Controller=? -1, Operator=0, SignalSource=ALab_CellC_v1.0_4 5362
EventTableTriggerIO 9289: IOValue=[1], IRC5Controller=? -1, Operator=0, SignalSource=ALab_CellC_v1.0_4 5362
EventTableTriggerIO 9290: IOValue=[0], IRC5Controller=? -1, Operator=0, SignalSource=ALab_CellC_v1.0_4 5362
EventTableTriggerIO 9291: IOValue=[0], IRC5Controller=? -1, Operator=0, SignalSource=ALab_CellC_v1.0_4 5362
EventTableTriggerIO 9292: IOValue=[1], IRC5Controller=? -1, Operator=0, SignalSource=ALab_CellC_v1.0_4 5362
EventTableTriggerIO 9293: IOValue=[1], IRC5Controller=? -1, Operator=0, SignalSource=ALab_CellC_v1.0_4 5362
EventTableTriggerIO 9294: IOValue=[0], IRC5Controller=? -1, Operator=0, SignalSource=ALab_CellC_v1.0_4 5362
EventTableTriggerIO 9295: IOValue=[1], IRC5Controller=? -1, Operator=0, SignalSource=LCFA_profile 1
EventTableTriggerIO 9296: IOValue=[1], IRC5Controller=? -1, Operator=0, SignalSource=LCFA_profile 1
EventTableTriggerIO 9297: IOValue=[1], IRC5Controller=? -1, Operator=0, SignalSource=ALab_CellC_v1.0_4 5362
EventTableTriggerIO 9298: IOValue=[0], IRC5Controller=? -1, Operator=0, SignalSource=ALab_CellC_v1.0_4 5362
EventTableTriggerIO 9299: IOValue=[1], IRC5Controller=? -1, Operator=0, SignalSource=ALab_CellC_v1.0_4 5362
EventTableTriggerIO 9300: IOValue=[0], IRC5Controller=? -1, Operator=0, SignalSource=ALab_CellC_v1.0_4 5362
EventTableTriggerLogic 9301: layoutX=167, layoutY=76, Operand1=AND 4076, Operand2=AND 4081, Operator=0, Delay=1000
EventTableTriggerLogic 9302: layoutX=194, layoutY=70, Operand1=AND 4088, Operand2=AND 4093, Operator=0, Delay=1000
EventTableTriggerLogic 9303: layoutX=181, layoutY=88, Operand1=AND 4100, Operand2=AND 4105, Operator=0, Delay=1000
EventTableTriggerLogic 9304: layoutX=165, layoutY=70, Operand1=AND 4112, Operand2=AND 4117, Operator=0, Delay=1000
EventTableTriggerLogic 9305: layoutX=217, layoutY=77, Operand1=AND 4123, Operand2=AND 4127, Operator=0, Delay=1000
EventTableTriggerLogic 9306: layoutX=168, layoutY=84, Operand1=AND 4135, Operand2=AND 4139, Operator=0, Delay=1000
EventTableTriggerLogic 9307: layoutX=219, layoutY=73, Operand1=AND 4146, Operand2=AND 4150, Operator=0, Delay=1000
EventTableTriggerLogic 9308: layoutX=203, layoutY=67, Operand1=AND 4157, Operand2=AND 4161, Operator=0, Delay=1000
EventTableTriggerLogic 9309: layoutX=220, layoutY=69, Operand1=AND 4167, Operand2=AND 4171, Operator=0, Delay=1000
EventTableTriggerLogic 9310: layoutX=243, layoutY=55, Operand1=AND 4179, Operand2=AND 4183, Operator=0, Delay=1000
EventTableTriggerLogic 9311: layoutX=204, layoutY=112, Operand1=AND 4190, Operand2=AND 4194, Operator=0, Delay=1000
EventTableTriggerLogic 9312: layoutX=245, layoutY=97, Operand1=AND 4201, Operand2=AND 4205, Operator=0, Delay=1000
EventTableTriggerLogic 9313: layoutX=234, layoutY=61, Operand1=AND 4211, Operand2=AND 4214, Operator=0, Delay=1000
EventTableTriggerLogic 9314: layoutX=192, layoutY=87, Operand1=AND 4222, Operand2=AND 4225, Operator=0, Delay=1000
EventTableTriggerLogic 9315: layoutX=212, layoutY=64, Operand1=AND 4232, Operand2=AND 4235, Operator=0, Delay=1000
EventTableTriggerLogic 9316: layoutX=160, layoutY=73, Operand1=AND 4242, Operand2=AND 4245, Operator=0, Delay=1000
EventTableTriggerLogic 9317: layoutX=153, layoutY=73, Operand1=AND 4264, Operand2=NOT 4269, Operator=0, Delay=1000
EventTableTriggerLogic 9318: layoutX=133, layoutY=81, Operand1=AND 4274, Operand2=conv1_buffer_upper_go_down 6332, Operator=0, Delay=1000
EventTableTriggerLogic 9319: layoutX=184, layoutY=91, Operand1=AND 4283, Operand2=NOT 4287, Operator=0, Delay=1000
EventTableTriggerLogic 9320: layoutX=211, layoutY=90, Operand1=AND 4292, Operand2=conv1_buffer_upper_go_down 6282, Operator=0, Delay=1000
EventTableTriggerLogic 9321: layoutX=226, layoutY=110, Operand1=AND 4300, Operand2=NOT 4304, Operator=0, Delay=1000
EventTableTriggerLogic 9322: layoutX=164, layoutY=68, Operand1=AND 4309, Operand2=conv1_buffer_upper_go_down 6288, Operator=0, Delay=1000
EventTableTriggerLogic 9323: layoutX=161, layoutY=63, Operand1=AND 4317, Operand2=NOT 4320, Operator=0, Delay=1000
EventTableTriggerLogic 9324: layoutX=174, layoutY=87, Operand1=AND 4325, Operand2=conv1_buffer_upper_go_down 6294, Operator=0, Delay=1000
EventTableTriggerLogic 9325: layoutX=148, layoutY=98, Operand1=AND 4332, Operand2=NOT 4337, Operator=0, Delay=1000
EventTableTriggerLogic 9326: layoutX=206, layoutY=74, Operand1=AND 4342, Operand2=conv2_buffer_upper_vertical_move 6300, Operator=0, Delay=1000
EventTableTriggerLogic 9327: layoutX=195, layoutY=82, Operand1=AND 4351, Operand2=NOT 4355, Operator=0, Delay=1000
EventTableTriggerLogic 9328: layoutX=193, layoutY=94, Operand1=AND 4360, Operand2=conv2_buffer_upper_vertical_move 6306, Operator=0, Delay=1000
EventTableTriggerLogic 9329: layoutX=210, layoutY=27, Operand1=conv2_buffer_horizontal_move 6309, Operand2=AND 4369, Operator=0, Delay=1000
EventTableTriggerLogic 9330: layoutX=233, layoutY=95, Operand1=AND 4377, Operand2=conv2_buffer_upper_vertical_move 6312, Operator=0, Delay=1000
EventTableTriggerLogic 9331: layoutX=102, layoutY=69, Operand1=AND 4385, Operand2=NOT 4388, Operator=0, Delay=1000
EventTableTriggerLogic 9332: layoutX=97, layoutY=92, Operand1=AND 4393, Operand2=conv2_buffer_upper_vertical_move 6318, Operator=0, Delay=1000
EventTableTriggerLogic 9333: layoutX=96, layoutY=16, Operand1=cellC_pallet_holder 7125, Operand2=cellC_pallet_stopper 7126, Operator=0, Delay=1000
EventTableTriggerLogic 9334: layoutX=142, layoutY=32, Operand1=NOT 7128, Operand2=cellC_pallet_stopper 7127, Operator=0, Delay=1000
EventTableTriggerLogic 9335: layoutX=51, layoutY=46, Operand1=NOT 7130, Operand2=NOT 7132, Operator=0, Delay=1000
EventTableTriggerLogic 9336: layoutX=107, layoutY=60, Operand1=cellC_pallet_holder 7134, Operand2=NOT 7135, Operator=0, Delay=1000
EventTableTriggerIO 9337: IOValue=[1], IRC5Controller=? -1, Operator=0, SignalSource=ALab_CellC_v1.0_4 5362
EventTableTriggerLogic 9338: layoutX=184, layoutY=128, Operand1=AND 6402, Operand2=AND 6408, Operator=0, Delay=1000
EventTableTriggerLogic 9339: layoutX=231, layoutY=144, Operand1=AND 6416, Operand2=pallet1 6426, Operator=0, Delay=1000
EventTableTriggerLogic 9340: layoutX=251, layoutY=143, Operand1=AND 8115, Operand2=pallet3.1 8114, Operator=0, Delay=1000
EventTableTriggerLogic 9341: layoutX=62, layoutY=38, Operand1=pallet2 8126, Operand2=cellC_slider_horizontal_move 8125, Operator=0, Delay=1000
EventTableTriggerLogic 9342: layoutX=133, layoutY=37, Operand1=pallet3 6451, Operand2=pose6 6452, Operator=0, Delay=1000
EventTableTriggerLogic 9343: layoutX=61, layoutY=50, Operand1=pallet3.2 6456, Operand2=pose3 6457, Operator=0, Delay=1000
EventTableTriggerLogic 9344: layoutX=131, layoutY=52, Operand1=pickpallet1 6461, Operand2=pose7 6462, Operator=0, Delay=1000
EventTableTriggerLogic 9345: layoutX=8, layoutY=16, Operand1=pickpallet2 6466, Operand2=pose13 6467, Operator=0, Delay=1000
EventTableTriggerLogic 9346: layoutX=232, layoutY=117, Operand1=AND 6471, Operand2=pallet4 6481, Operator=0, Delay=1000
EventTableTriggerLogic 9347: layoutX=237, layoutY=122, Operand1=AND 6485, Operand2=conv2_buffer_stopper 6492, Operator=0, Delay=1000
EventTableTriggerLogic 9348: layoutX=240, layoutY=90, Operand1=AND 6496, Operand2=AND 6500, Operator=0, Delay=1000
EventTableTriggerLogic 9349: layoutX=80, layoutY=49, Operand1=pallet5.1 6513, Operand2=conv2_outer_lifter 6514, Operator=0, Delay=1000
EventTableTriggerIO 9350: IOValue=[1], IRC5Controller=? -1, Operator=0, SignalSource=LCFA_profile 1
EventTableTriggerIO 9351: IOValue=[1], IRC5Controller=? -1, Operator=0, SignalSource=LCFA_profile 1
EventTableTriggerIO 9352: IOValue=[1], IRC5Controller=? -1, Operator=0, SignalSource=LCFA_profile 1
EventTableTriggerIO 9353: IOValue=[1], IRC5Controller=? -1, Operator=0, SignalSource=LCFA_profile 1
EventTableTriggerIO 9354: IOValue=[1], IRC5Controller=? -1, Operator=0, SignalSource=LCFA_profile 1
EventTableTriggerIO 9355: IOValue=[1], IRC5Controller=? -1, Operator=0, SignalSource=LCFA_profile 1
EventTableTriggerIO 9356: IOValue=[1], IRC5Controller=? -1, Operator=0, SignalSource=LCFA_profile 1
EventTableTriggerIO 9357: IOValue=[1], IRC5Controller=? -1, Operator=0, SignalSource=LCFA_profile 1
EventTableTriggerIO 9358: IOValue=[1], IRC5Controller=? -1, Operator=0, SignalSource=LCFA_profile 1
EventTableTriggerIO 9359: IOValue=[1], IRC5Controller=? -1, Operator=0, SignalSource=LCFA_profile 1
EventTableTriggerIO 9360: IOValue=[0], IRC5Controller=? -1, Operator=0, SignalSource=ALab_CellC_v1.0_4 5362
EventTableTriggerIO 9361: IOValue=[1], IRC5Controller=? -1, Operator=0, SignalSource=ALab_CellC_v1.0_4 5362
EventTableTriggerIO 9362: IOValue=[0], IRC5Controller=? -1, Operator=0, SignalSource=ALab_CellC_v1.0_4 5362
EventTableTriggerIO 9363: IOValue=[1], IRC5Controller=? -1, Operator=0, SignalSource=ALab_CellC_v1.0_4 5362
EventTableTriggerIO 9364: IOValue=[1], IRC5Controller=? -1, Operator=0, SignalSource=ALab_CellC_v1.0_4 5362
EventTableTriggerIO 9365: IOValue=[0], IRC5Controller=? -1, Operator=0, SignalSource=ALab_CellC_v1.0_4 5362
EventTableTriggerIO 9366: IOValue=[0], IRC5Controller=? -1, Operator=0, SignalSource=ALab_CellC_v1.0_4 5362
EventTableTriggerIO 9367: IOValue=[1], IRC5Controller=? -1, Operator=0, SignalSource=ALab_CellC_v1.0_4 5362
EventTableTriggerIO 9368: IOValue=[1], IRC5Controller=? -1, Operator=0, SignalSource=ALab_CellC_v1.0_4 5362
EventTableTriggerIO 9369: IOValue=[0], IRC5Controller=? -1, Operator=0, SignalSource=ALab_CellC_v1.0_4 5362
EventTableTriggerIO 9370: IOValue=[1], IRC5Controller=? -1, Operator=0, SignalSource=ALab_CellC_v1.0_4 5362
EventTableTriggerIO 9371: IOValue=[0], IRC5Controller=? -1, Operator=0, SignalSource=ALab_CellC_v1.0_4 5362
EventTableTriggerIO 9372: IOValue=[0], IRC5Controller=? -1, Operator=0, SignalSource=ALab_CellC_v1.0_4 5362
EventTableTriggerIO 9373: IOValue=[1], IRC5Controller=? -1, Operator=0, SignalSource=ALab_CellC_v1.0_4 5362
EventTableTriggerIO 9374: IOValue=[1], IRC5Controller=? -1, Operator=0, SignalSource=ALab_CellC_v1.0_4 5362
EventTableTriggerIO 9375: IOValue=[0], IRC5Controller=? -1, Operator=0, SignalSource=ALab_CellC_v1.0_4 5362
EventTableTriggerIO 9376: IOValue=[0], IRC5Controller=? -1, Operator=0, SignalSource=ALab_CellC_v1.0_4 5362
EventTableTriggerIO 9377: IOValue=[1], IRC5Controller=? -1, Operator=0, SignalSource=ALab_CellC_v1.0_4 5362
EventTableTriggerIO 9378: IOValue=[1], IRC5Controller=? -1, Operator=0, SignalSource=ALab_CellC_v1.0_4 5362
EventTableTriggerIO 9379: IOValue=[0], IRC5Controller=? -1, Operator=0, SignalSource=ALab_CellC_v1.0_4 5362
EventTableTriggerIO 9380: IOValue=[1], IRC5Controller=? -1, Operator=0, SignalSource=LCFA_profile 1
EventTableTriggerIO 9381: IOValue=[1], IRC5Controller=? -1, Operator=0, SignalSource=LCFA_profile 1
EventTableTriggerIO 9382: IOValue=[1], IRC5Controller=? -1, Operator=0, SignalSource=LCFA_profile 1
EventTableTriggerIO 9383: IOValue=[1], IRC5Controller=? -1, Operator=0, SignalSource=LCFA_profile 1
EventTableTriggerIO 9384: IOValue=[1], IRC5Controller=? -1, Operator=0, SignalSource=ALab_CellC_v1.0_4 5362
EventTableTriggerIO 9385: IOValue=[0], IRC5Controller=? -1, Operator=0, SignalSource=ALab_CellC_v1.0_4 5362
EventTableTriggerIO 9386: IOValue=[1], IRC5Controller=? -1, Operator=0, SignalSource=LCFA_profile 1
EventTableTriggerIO 9387: IOValue=[1], IRC5Controller=? -1, Operator=0, SignalSource=LCFA_profile 1
EventTableTriggerIO 9388: IOValue=[1], IRC5Controller=? -1, Operator=0, SignalSource=LCFA_profile 1
EventTableTriggerIO 9389: IOValue=[1], IRC5Controller=? -1, Operator=0, SignalSource=LCFA_profile 1
EventTableTriggerIO 9390: IOValue=[1], IRC5Controller=? -1, Operator=0, SignalSource=ALab_CellC_v1.0_4 5362
EventTableTriggerIO 9391: IOValue=[0], IRC5Controller=? -1, Operator=0, SignalSource=ALab_CellC_v1.0_4 5362
EventTableTriggerIO 9392: IOValue=[1], IRC5Controller=? -1, Operator=0, SignalSource=ALab_CellC_v1.0_4 5362
EventTableTriggerIO 9393: IOValue=[0], IRC5Controller=? -1, Operator=0, SignalSource=ALab_CellC_v1.0_4 5362
EventTableTriggerIO 9394: IOValue=[0], IRC5Controller=? -1, Operator=0, SignalSource=ALab_CellC_v1.0_4 5362
EventTableTriggerIO 9395: IOValue=[1], IRC5Controller=? -1, Operator=0, SignalSource=ALab_CellC_v1.0_4 5362
EventTableTriggerIO 9396: IOValue=[1], IRC5Controller=? -1, Operator=0, SignalSource=ALab_CellC_v1.0_4 5362
EventTableTriggerIO 9397: IOValue=[0], IRC5Controller=? -1, Operator=0, SignalSource=ALab_CellC_v1.0_4 5362
EventTableTriggerIO 9398: IOValue=[1], IRC5Controller=? -1, Operator=0, SignalSource=LCFA_profile 1
EventTableTriggerIO 9399: IOValue=[1], IRC5Controller=? -1, Operator=0, SignalSource=LCFA_profile 1
EventTableTriggerIO 9400: IOValue=[1], IRC5Controller=? -1, Operator=0, SignalSource=LCFA_profile 1
EventTableTriggerLogic 9401: layoutX=150, layoutY=90, Operand1=AND 6770, Operand2=conv2_motor_s1 6766, Operator=0, Delay=1000
EventTableTriggerIO 9402: IOValue=[1], IRC5Controller=? -1, Operator=0, SignalSource=LCFA_profile 1
EventTableTriggerIO 9403: IOValue=[1], IRC5Controller=? -1, Operator=0, SignalSource=LCFA_profile 1
EventTableTriggerIO 9404: IOValue=[1], IRC5Controller=? -1, Operator=0, SignalSource=LCFA_profile 1
EventTableTriggerIO 9405: IOValue=[1], IRC5Controller=? -1, Operator=0, SignalSource=LCFA_profile 1
EventTableTriggerIO 9406: IOValue=[1], IRC5Controller=? -1, Operator=0, SignalSource=LCFA_profile 1
EventTableTriggerIO 9407: IOValue=[1], IRC5Controller=? -1, Operator=0, SignalSource=LCFA_profile 1
EventTableTriggerIO 9408: IOValue=[1], IRC5Controller=? -1, Operator=0, SignalSource=LCFA_profile 1
EventTableTriggerIO 9409: IOValue=[1], IRC5Controller=? -1, Operator=0, SignalSource=LCFA_profile 1
EventTableTriggerIO 9410: IOValue=[1], IRC5Controller=? -1, Operator=0, SignalSource=LCFA_profile 1
EventTableTriggerIO 9411: IOValue=[1], IRC5Controller=? -1, Operator=0, SignalSource=LCFA_profile 1
EventTableTriggerIO 9412: IOValue=[1], IRC5Controller=? -1, Operator=0, SignalSource=LCFA_profile 1
EventTableTriggerIO 9413: IOValue=[1], IRC5Controller=? -1, Operator=0, SignalSource=LCFA_profile 1
EventTableTriggerLogic 9414: layoutX=155, layoutY=137, Operand1=AND 6751, Operand2=NOT 6755, Operator=0, Delay=1000
EventTableTriggerIO 9415: IOValue=[1], IRC5Controller=? -1, Operator=0, SignalSource=LCFA_profile 1
EventTableTriggerIO 9416: IOValue=[1], IRC5Controller=? -1, Operator=0, SignalSource=LCFA_profile 1
EventTableTriggerLogic 9417: layoutX=48, layoutY=41, Operand1=pallet1.1 6778, Operand2=PalletIO00 6779, Operator=0, Delay=1000
EventTableTriggerIO 9418: IOValue=[1], IRC5Controller=? -1, Operator=0, SignalSource=LCFA_profile 1
EventTableTriggerIO 9419: IOValue=[1], IRC5Controller=? -1, Operator=0, SignalSource=ALab_CellC_v1.0_4 5362
EventTableTriggerIO 9420: IOValue=[0], IRC5Controller=? -1, Operator=0, SignalSource=ALab_CellC_v1.0_4 5362
EventTableTriggerLogic 9421: layoutX=103, layoutY=47, Operand1=NOT 8291, Operand2=pallet5 8290, Operator=0, Delay=1000
EventTableTriggerLogic 9422: layoutX=79, layoutY=37, Operand1=Pallet5.3 8029, Operand2=conv2_buffer_upper_vertical_move 8133, Operator=0, Delay=1000
EventTableTriggerLogic 9423: layoutX=40, layoutY=37, Operand1=Pallet5.4 8035, Operand2=conv2_buffer_lower_vertical_move 8036, Operator=0, Delay=1000
EventTableTriggerLogic 9424: layoutX=103, layoutY=47, Operand1=conv2_buffer_horizontal_move 8134, Operand2=Pallet5.7 8040, Operator=0, Delay=1000
EventTableTriggerLogic 9425: layoutX=54, layoutY=45, Operand1=NOT 8135, Operand2=Pallet5.6 8046, Operator=0, Delay=1000
EventTableTriggerLogic 9426: layoutX=108, layoutY=46, Operand1=NOT 8052, Operand2=Pallet5.5 8051, Operator=0, Delay=1000
EventTableTriggerIO 9427: IOValue=[1], IRC5Controller=? -1, Operator=0, SignalSource=LCFA_profile 1
EventTableTriggerIO 9428: IOValue=[1], IRC5Controller=? -1, Operator=0, SignalSource=LCFA_profile 1
EventTableTriggerIO 9429: IOValue=[1], IRC5Controller=? -1, Operator=0, SignalSource=LCFA_profile 1
EventTableTriggerIO 9430: IOValue=[1], IRC5Controller=? -1, Operator=0, SignalSource=LCFA_profile 1
EventTableTriggerIO 9431: IOValue=[1], IRC5Controller=? -1, Operator=0, SignalSource=LCFA_profile 1
EventTableTriggerIO 9432: IOValue=[1], IRC5Controller=? -1, Operator=0, SignalSource=LCFA_profile 1
EventTableTriggerIO 9433: IOValue=[1], IRC5Controller=? -1, Operator=0, SignalSource=LCFA_profile 1
EventTableTriggerIO 9434: IOValue=[1], IRC5Controller=? -1, Operator=0, SignalSource=LCFA_profile 1
EventTableTriggerIO 9435: IOValue=[1], IRC5Controller=? -1, Operator=0, SignalSource=LCFA_profile 1
EventTableTriggerIO 9436: IOValue=[1], IRC5Controller=? -1, Operator=0, SignalSource=LCFA_profile 1
EventTableTriggerIO 9437: IOValue=[1], IRC5Controller=? -1, Operator=0, SignalSource=LCFA_profile 1
EventTableTriggerIO 9438: IOValue=[1], IRC5Controller=? -1, Operator=0, SignalSource=LCFA_profile 1
EventTableTriggerIO 9439: IOValue=[1], IRC5Controller=? -1, Operator=0, SignalSource=LCFA_profile 1
EventTableTriggerIO 9440: IOValue=[1], IRC5Controller=? -1, Operator=0, SignalSource=LCFA_profile 1
EventTableTriggerIO 9441: IOValue=[1], IRC5Controller=? -1, Operator=0, SignalSource=LCFA_profile 1
EventTableTriggerIO 9442: IOValue=[1], IRC5Controller=? -1, Operator=0, SignalSource=LCFA_profile 1
EventTableTriggerIO 9443: IOValue=[1], IRC5Controller=? -1, Operator=0, SignalSource=LCFA_profile 1
EventTableTriggerLogic 9444: layoutX=99, layoutY=32, Operand1=Pallet2.1 8141, Operand2=NOT 8139, Operator=0, Delay=1000
EventTableTriggerLogic 9445: layoutX=181, layoutY=52, Operand1=conv1_buffer_upper_go_down 8146, Operand2=Pallet2.2 8145, Operator=0, Delay=1000
EventTableTriggerLogic 9446: layoutX=48, layoutY=51, Operand1=Pallet2.3 8150, Operand2=conv1_buffer_lower_go_up 8151, Operator=0, Delay=1000
EventTableTriggerLogic 9447: layoutX=67, layoutY=33, Operand1=pallet2 8155, Operand2=NOT 8156, Operator=0, Delay=1000
EventTableTriggerLogic 9448: layoutX=102, layoutY=29, Operand1=Pallet2.4 8161, Operand2=NOT 8162, Operator=0, Delay=1000
EventTableTriggerLogic 9449: layoutX=102, layoutY=23, Operand1=Pallet2.5 8167, Operand2=NOT 8168, Operator=0, Delay=1000
EventTableTriggerIO 9450: IOValue=[1], IRC5Controller=? -1, Operator=0, SignalSource=LCFA_profile 1
EventTableTriggerIO 9451: IOValue=[1], IRC5Controller=? -1, Operator=0, SignalSource=LCFA_profile 1
EventTableTriggerIO 9452: IOValue=[1], IRC5Controller=? -1, Operator=0, SignalSource=LCFA_profile 1
EventTableTriggerIO 9453: IOValue=[1], IRC5Controller=? -1, Operator=0, SignalSource=LCFA_profile 1
EventTableTriggerIO 9454: IOValue=[1], IRC5Controller=? -1, Operator=0, SignalSource=LCFA_profile 1
EventTableTriggerIO 9455: IOValue=[1], IRC5Controller=? -1, Operator=0, SignalSource=LCFA_profile 1
EventTableTriggerIO 9456: IOValue=[1], IRC5Controller=? -1, Operator=0, SignalSource=LCFA_profile 1
EventTableTriggerIO 9457: IOValue=[1], IRC5Controller=? -1, Operator=0, SignalSource=LCFA_profile 1
EventTableTriggerIO 9458: IOValue=[1], IRC5Controller=? -1, Operator=0, SignalSource=LCFA_profile 1
EventTableTriggerIO 9459: IOValue=[1], IRC5Controller=? -1, Operator=0, SignalSource=LCFA_profile 1
EventTableTriggerIO 9460: IOValue=[1], IRC5Controller=? -1, Operator=0, SignalSource=LCFA_profile 1
EventTableTriggerIO 9461: IOValue=[1], IRC5Controller=? -1, Operator=0, SignalSource=LCFA_profile 1
EventTableTriggerIO 9462: IOValue=[1], IRC5Controller=? -1, Operator=0, SignalSource=LCFA_profile 1
EventTableTriggerLogic 9463: layoutX=49, layoutY=26, Operand1=Pallet2.6 8213, Operand2=conv1_buffer_horizontal_open 8214, Operator=0, Delay=1000
EventTableTriggerIO 9464: IOValue=[1], IRC5Controller=? -1, Operator=0, SignalSource=LCFA_profile 1
EventTableTriggerIO 9465: IOValue=[1], IRC5Controller=? -1, Operator=0, SignalSource=LCFA_profile 1
EventTableTriggerIO 9466: IOValue=[1], IRC5Controller=? -1, Operator=0, SignalSource=LCFA_profile 1
EventTableTriggerIO 9467: IOValue=[1], IRC5Controller=? -1, Operator=0, SignalSource=LCFA_profile 1
EventTableTriggerIO 9468: IOValue=[1], IRC5Controller=? -1, Operator=0, SignalSource=LCFA_profile 1
EventTableTriggerIO 9469: IOValue=[1], IRC5Controller=? -1, Operator=0, SignalSource=ALab_CellC_v1.0_4 5362
EventTableTriggerIO 9470: IOValue=[0], IRC5Controller=? -1, Operator=0, SignalSource=ALab_CellC_v1.0_4 5362
EventTableTriggerIO 9471: IOValue=[1], IRC5Controller=? -1, Operator=0, SignalSource=ALab_CellC_v1.0_4 5362
EventTableTriggerIO 9472: IOValue=[0], IRC5Controller=? -1, Operator=0, SignalSource=ALab_CellC_v1.0_4 5362
EventTableTriggerIO 9473: IOValue=[1], IRC5Controller=? -1, Operator=0, SignalSource=ALab_CellC_v1.0_4 5362
EventTableTriggerIO 9474: IOValue=[0], IRC5Controller=? -1, Operator=0, SignalSource=ALab_CellC_v1.0_4 5362
EventTableTriggerIO 9475: IOValue=[0], IRC5Controller=? -1, Operator=0, SignalSource=ALab_CellC_v1.0_4 5362
EventTableTriggerIO 9476: IOValue=[1], IRC5Controller=? -1, Operator=0, SignalSource=ALab_CellC_v1.0_4 5362
EventTableTriggerIO 9477: IOValue=[0], IRC5Controller=? -1, Operator=0, SignalSource=ALab_CellC_v1.0_4 5362
EventTableTriggerIO 9478: IOValue=[1], IRC5Controller=? -1, Operator=0, SignalSource=ALab_CellC_v1.0_4 5362
EventTableTriggerIO 9479: IOValue=[1], IRC5Controller=? -1, Operator=0, SignalSource=ALab_CellC_v1.0_4 5362
EventTableTriggerIO 9480: IOValue=[0], IRC5Controller=? -1, Operator=0, SignalSource=ALab_CellC_v1.0_4 5362
EventTableTriggerIO 9481: IOValue=[0], IRC5Controller=? -1, Operator=0, SignalSource=ALab_CellC_v1.0_4 5362
EventTableTriggerIO 9482: IOValue=[1], IRC5Controller=? -1, Operator=0, SignalSource=ALab_CellC_v1.0_4 5362
EventTableTriggerIO 9483: IOValue=[1], IRC5Controller=? -1, Operator=0, SignalSource=ALab_CellC_v1.0_4 5362
EventTableTriggerIO 9484: IOValue=[0], IRC5Controller=? -1, Operator=0, SignalSource=ALab_CellC_v1.0_4 5362
EventTableTriggerIO 9485: IOValue=[0], IRC5Controller=? -1, Operator=0, SignalSource=ALab_CellC_v1.0_4 5362
EventTableTriggerIO 9486: IOValue=[1], IRC5Controller=? -1, Operator=0, SignalSource=ALab_CellC_v1.0_4 5362
EventTableTriggerIO 9487: IOValue=[1], IRC5Controller=? -1, Operator=0, SignalSource=ALab_CellC_v1.0_4 5362
EventTableTriggerIO 9488: IOValue=[0], IRC5Controller=? -1, Operator=0, SignalSource=ALab_CellC_v1.0_4 5362
EventTableTriggerIO 9489: IOValue=[1], IRC5Controller=? -1, Operator=0, SignalSource=LCFA_profile 1
EventTableTriggerIO 9490: IOValue=[1], IRC5Controller=? -1, Operator=0, SignalSource=LCFA_profile 1
EventTableTriggerIO 9491: IOValue=[1], IRC5Controller=? -1, Operator=0, SignalSource=ALab_CellC_v1.0_4 5362
EventTableTriggerIO 9492: IOValue=[0], IRC5Controller=? -1, Operator=0, SignalSource=ALab_CellC_v1.0_4 5362
EventTableTriggerIO 9493: IOValue=[1], IRC5Controller=? -1, Operator=0, SignalSource=ALab_CellC_v1.0_4 5362
EventTableTriggerIO 9494: IOValue=[0], IRC5Controller=? -1, Operator=0, SignalSource=ALab_CellC_v1.0_4 5362
Station logic (signal -> signal, property => property):
  ALab_CellC_v1.0_4.Rob1_Gripper_Reset -> Rubic Cube Simulation .DI_Open
  ALab_CellC_v1.0_4.Rob1_Gripper_Set -> Rubic Cube Simulation .DI_Close
Targets, tools, work objects and paths stored in the station and not in the controller backup, written as RAPID:
! task T_ROB1
MODULE MainModule
  CONST robtarget Target_10:=[[419.99,-377.933,712],[0.707106781,0,0,-0.707106781],[0,0,0,0],[9E+09,9E+09,9E+09,9E+09,9E+09,9E+09]];
ENDMODULE


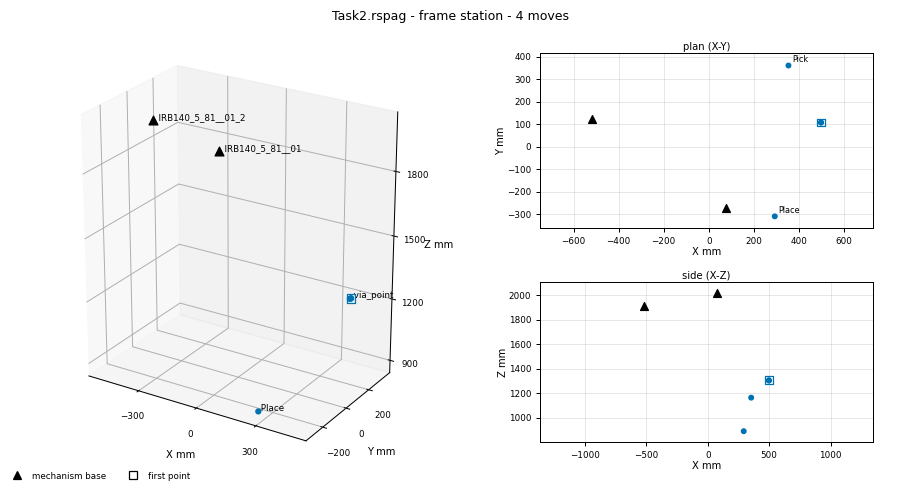
[picture p0: tool path of Task2.rspag in frame station, 4 of 9 moves have a stored position in this frame; points joined in program order, loops and branches not executed]
--- Backups/ALab_CellC_v1.0_4/RAPID/TASK1/PROGMOD/CalibData.mod ---
MODULE CalibData
    PERS tooldata Fingers:=[TRUE,[[0,0,50],[1,0,0,0]],[1,[0,0,1],[1,0,0,0],0,0,0]];
ENDMODULE

--- Backups/ALab_CellC_v1.0_4/RAPID/TASK1/PROGMOD/MainModule.mod ---
MODULE MainModule
    CONST robtarget via_point:=[[419.99,-377.933,712],[0.707106781,0,0,-0.707106781],[0,0,0,0],[9E+09,9E+09,9E+09,9E+09,9E+09,9E+09]];
    CONST robtarget Pick:=[[275.502,-630.736,852.224],[0.707106781,0,0,-0.707106781],[0,0,0,0],[9E+09,9E+09,9E+09,9E+09,9E+09,9E+09]];
    CONST robtarget Place:=[[214.792273259,38.46617002,1125.252179854],[0.707106922,0.000000191,0.000000183,-0.70710664],[0,2,0,0],[9E+09,9E+09,9E+09,9E+09,9E+09,9E+09]];

    PROC main()
        HomePosition;
        Path_10;            !routinre for pick and place
        HomePosition;

    ENDPROC


    PROC HomePosition()
		MoveAbsJ [[0,0,0,0,0,0],[9E+09,9E+09,9E+09,9E+09,9E+09,9E+09]]\NoEOffs,v200,z50,tool0;
	ENDPROC

    !Function for closing gripper
    PROC CloseGripper()
        SetDO Rob1_Gripper_Reset,0;
        SetDO Rob1_Gripper_Set,1;
        WaitDO Rob1_Gripper_Set,1;
        WaitTime 1;
    ENDPROC

    !Function for opening gripper
    PROC OpenGripper()
        SetDO Rob1_Gripper_Set,0;
        SetDO Rob1_Gripper_Reset,1;
        WaitDO Rob1_Gripper_Reset,1;
        WaitTime 1;
    ENDPROC

    PROC Path_10()
        VAR robtarget PrePick; !declearing variable for creating offset
        VAR robtarget PrePlace; !declearing variable for creating offset

        PrePick:=Offs(Pick, 0, 0, -100); ! creating offset from the pick point
        PrePlace:=Offs(Place, 0, 0,-100); ! creating offset from the place point


        OpenGripper;

        !via point
        MoveJ via_point,v500,z0,Fingers\WObj:=wobj0;

        ! going to the pick point
        MoveJ PrePick,v500,z0,Fingers\WObj:=wobj0;
        MoveL Pick,v50,fine,Fingers\WObj:=wobj0;
        WaitRob \ZeroSpeed;

        CloseGripper;

        MoveL PrePick,v50,fine,Fingers\WObj:=wobj0;

        !via point
        MoveJ via_point,v500,z0,Fingers\WObj:=wobj0;

        ! going to the place point
        MoveJ PrePlace,v500,z0,Fingers\WObj:=wobj0;
        MoveL Place,v50,fine,Fingers\WObj:=wobj0;
        WaitRob \ZeroSpeed;
        OpenGripper;


    ENDPROC

ENDMODULE

--- Backups/ALab_CellC_v1.0_4/RAPID/TASK2/PROGMOD/CalibData.mod ---
MODULE CalibData
	TASK PERS wobjdata Wobjmytool:=[TRUE,TRUE,"",[[0,0,0],[1,0,0,0]],[[0,0,0],[1,0,0,0]]];
ENDMODULE

--- Backups/ALab_CellC_v1.0_4/RAPID/TASK2/PROGMOD/MainModule.mod ---
MODULE MainModule

    PROC main()
        HomePosition;

        ! Value "1" sets on the Digital Output
        ! Value "0" sets off the Digital Output


    ENDPROC

    PROC HomePosition()
		MoveAbsJ [[0,0,0,0,0,0],[9E+09,9E+09,9E+09,9E+09,9E+09,9E+09]]\NoEOffs,v200,z50,tool0;
	ENDPROC
ENDMODULE

--- Backups/ALab_CellC_v1.0_4/SYSPAR/EIO.cfg ---
EIO:CFG_1.0:5:0::
#
EIO_BUS:

      -Name "Virtual1" -ConnectorID "SIM1"

      -Name "DeviceNet1" -BusType "DNET" -ConnectorID "PCI1"\
      -ConnectorLabel "First DeviceNet"

      -Name "DeviceNet2" -BusType "DNET" -ConnectorID "PCI2"\
      -ConnectorLabel "Second DeviceNet" -DN_MasterAddress 1
#
EIO_UNIT_TYPE:

      -Name "Virtual" -VendorName "ABB" -ProductName "Virtual unit"

      -Name "DN_GENERIC" -BusType "DNET" -DN_ExplicitMsgEnabled \
      -DN_C1OutputSize -1 -DN_C1InputSize -1

      -Name "d320" -BusType "DNET" -VendorName "ABB Robotics"\
      -ProductName "120 Vac Unit" -DN_VendorId 75 -DN_ProductCode 1\
      -DN_DeviceType 7 -DN_MajorRev 1 -DN_ExplicitMsgEnabled  -DN_C1Interval 50\
      -DN_C1OutputSize 2 -DN_C1InputSize 2

      -Name "d327" -BusType "DNET" -VendorName "ABB Robotics"\
      -ProductName "Combi Unit" -DN_VendorId 75 -DN_ProductCode 2\
      -DN_DeviceType 100 -DN_MajorRev 5 -DN_ExplicitMsgEnabled \
      -DN_C1Interval 50 -DN_C1OutputSize 6 -DN_C1InputSize 2

      -Name "d328" -BusType "DNET" -VendorName "ABB Robotics"\
      -ProductName "24 VDC Unit" -DN_VendorId 75 -DN_ProductCode 3\
      -DN_DeviceType 7 -DN_ExplicitMsgEnabled  -DN_C1Interval 50\
      -DN_C1OutputSize 2 -DN_C1InputSize 2

      -Name "d332" -BusType "DNET" -VendorName "ABB Robotics"\
      -ProductName "Relay Unit" -DN_VendorId 75 -DN_ProductCode 5\
      -DN_DeviceType 7 -DN_MajorRev 2 -DN_ExplicitMsgEnabled  -DN_C1Interval 50\
      -DN_C1OutputSize 2 -DN_C1InputSize 2

      -Name "d327A" -BusType "DNET" -VendorName "ABB Robotics"\
      -ProductName "Combi Unit" -DN_VendorId 75 -DN_ProductCode 2\
      -DN_DeviceType 100 -DN_MajorRev 5 -DN_ExplicitMsgEnabled  -DN_C1Type "COS"\
      -DN_C1OutputSize 6 -DN_C1InputSize 2

      -Name "d328A" -BusType "DNET" -VendorName "ABB Robotics"\
      -ProductName "24 VDC Unit" -DN_VendorId 75 -DN_ProductCode 3\
      -DN_DeviceType 7 -DN_ExplicitMsgEnabled  -DN_C1Type "COS"\
      -DN_C1OutputSize 2 -DN_C1InputSize 2

      -Name "d332A" -BusType "DNET" -VendorName "ABB Robotics"\
      -ProductName "Relay Unit" -DN_VendorId 75 -DN_ProductCode 5\
      -DN_DeviceType 7 -DN_MajorRev 2 -DN_ExplicitMsgEnabled  -DN_C1Type "COS"\
      -DN_C1OutputSize 2 -DN_C1InputSize 2

      -Name "d355A" -BusType "DNET" -VendorName "ABB Robotics"\
      -ProductName "Analog Unit" -DN_VendorId 75 -DN_ProductCode 10\
      -DN_DeviceType 100 -DN_MajorRev 1 -DN_ExplicitMsgEnabled \
      -DN_C1Interval 50 -DN_C1OutputSize 8 -DN_C1InputSize 8

